LIN {X 0,Y 431.74,Z 953.951,A -85,B 0,C 180,E1 3788.335,E2 3788.335} C_VEL
LIN {X 0,Y 438.13,Z 926.777,A -85,B 0,C 180,E1 3787.877,E2 3787.877} C_VEL
LIN {X 0,Y 442.587,Z 899.79,A -85,B 0,C 180,E1 3787.482,E2 3787.482} C_VEL
LIN {X 0,Y 459.904,Z 746.935,A -85,B 0,C 180,E1 3785.438,E2 3785.438} C_VEL
LIN {X 0,Y 462.106,Z 727.315,A -85,B 0,C 180,E1 3785.152,E2 3785.152} C_VEL
LIN {X 0,Y 460.748,Z 722.782,A -85,B 0,C 180,E1 3780.497,E2 3780.497} C_VEL
LIN {X 0,Y 460.764,Z 722.91,A -85,B 0,C 180,E1 3779.005,E2 3779.005} C_VEL
LIN {X 0,Y 462.101,Z 727.286,A -85,B 0,C 180,E1 3774.661,E2 3774.661} C_VEL
LIN {X 0,Y 442.705,Z 898.388,A -85,B 0,C 180,E1 3772.376,E2 3772.376} C_VEL
LIN {X 0,Y 438.374,Z 924.66,A -85,B 0,C 180,E1 3771.993,E2 3771.993} C_VEL
LIN {X 0,Y 432.03,Z 951.964,A -85,B 0,C 180,E1 3771.518,E2 3771.518} C_VEL
LIN {X 0,Y 425.902,Z 973.345,A -85,B 0,C 180,E1 3771.046,E2 3771.046} C_VEL
LIN {X 0,Y 419.197,Z 993.326,A -85,B 0,C 180,E1 3770.513,E2 3770.513} C_VEL
LIN {X 0,Y 411.382,Z 1013.618,A -85,B 0,C 180,E1 3769.866,E2 3769.866} C_VEL
LIN {X 0,Y 401.355,Z 1036.487,A -85,B 0,C 180,E1 3768.989,E2 3768.989} C_VEL
LIN {X 0,Y 388.724,Z 1061.334,A -85,B 0,C 180,E1 3767.816,E2 3767.816} C_VEL
LIN {X 0,Y 378.046,Z 1080.059,A -85,B 0,C 180,E1 3766.742,E2 3766.742} C_VEL
LIN {X 0,Y 367.06,Z 1097.609,A -85,B 0,C 180,E1 3765.565,E2 3765.565} C_VEL
LIN {X 0,Y 355.375,Z 1114.731,A -85,B 0,C 180,E1 3764.215,E2 3764.215} C_VEL
LIN {X 0,Y 342.365,Z 1132.293,A -85,B 0,C 180,E1 3762.566,E2 3762.566} C_VEL
LIN {X 0,Y 325.314,Z 1153.259,A -85,B 0,C 180,E1 3760.147,E2 3760.147} C_VEL
LIN {X 0,Y 310.967,Z 1169.357,A -85,B 0,C 180,E1 3757.833,E2 3757.833} C_VEL
LIN {X 0,Y 297.909,Z 1183.077,A -85,B 0,C 180,E1 3755.454,E2 3755.454} C_VEL
LIN {X 0,Y 284.669,Z 1196.186,A -85,B 0,C 180,E1 3752.712,E2 3752.712} C_VEL
LIN {X 0,Y 270.089,Z 1209.874,A -85,B 0,C 180,E1 3749.198,E2 3749.198} C_VEL
LIN {X 0,Y 254.111,Z 1223.984,A -85,B 0,C 180,E1 3744.547,E2 3744.547} C_VEL
LIN {X 0,Y 242.024,Z 1234.259,A -85,B 0,C 180,E1 3740.221,E2 3740.221} C_VEL
LIN {X 0,Y 231.488,Z 1243.083,A -85,B 0,C 180,E1 3735.593,E2 3735.593} C_VEL
LIN {X 0,Y 221.707,Z 1251.328,A -85,B 0,C 180,E1 3730.167,E2 3730.167} C_VEL
LIN {X 0,Y 211.776,Z 1260.022,A -85,B 0,C 180,E1 3722.572,E2 3722.572} C_VEL
LIN {X 0,Y 206.37,Z 1265.193,A -85,B 0,C 180,E1 3716.479,E2 3716.479} C_VEL
LIN {X 0,Y 202.92,Z 1269.061,A -85,B 0,C 180,E1 3710.486,E2 3710.486} C_VEL
LIN {X 0,Y 200.916,Z 1271.91,A -85,B 0,C 180,E1 3704.416,E2 3704.416} C_VEL
LIN {X 0,Y 200.12,Z 1273.63,A -85,B 0,C 180,E1 3698.918,E2 3698.918} C_VEL
LIN {X 0,Y 199.932,Z 1274.524,A -85,B 0,C 180,E1 3693.736,E2 3693.736} C_VEL
LIN {X 0,Y 199.902,Z 1274.714,A -85,B 0,C 180,E1 3688.575,E2 3688.575} C_VEL
LIN {X 0,Y 200.031,Z 1274.064,A -85,B 0,C 180,E1 3682.83,E2 3682.83} C_VEL
LIN {X 0,Y 200.717,Z 1272.303,A -85,B 0,C 180,E1 3676.468,E2 3676.468} C_VEL
LIN {X 0,Y 202.505,Z 1269.613,A -85,B 0,C 180,E1 3670.391,E2 3670.391} C_VEL
LIN {X 0,Y 205.725,Z 1265.905,A -85,B 0,C 180,E1 3664.38,E2 3664.38} C_VEL
LIN {X 0,Y 210.576,Z 1261.15,A -85,B 0,C 180,E1 3658.523,E2 3658.523} C_VEL
LIN {X 0,Y 217.466,Z 1255.015,A -85,B 0,C 180,E1 3652.644,E2 3652.644} C_VEL
LIN {X 0,Y 227.949,Z 1246.234,A -85,B 0,C 180,E1 3646.14,E2 3646.14} C_VEL
LIN {X 0,Y 240.257,Z 1235.835,A -85,B 0,C 180,E1 3640.408,E2 3640.408} C_VEL
LIN {X 0,Y 251.535,Z 1226.259,A -85,B 0,C 180,E1 3636.215,E2 3636.215} C_VEL
LIN {X 0,Y 263.975,Z 1215.419,A -85,B 0,C 180,E1 3632.378,E2 3632.378} C_VEL
LIN {X 0,Y 279.527,Z 1201.327,A -85,B 0,C 180,E1 3628.38,E2 3628.38} C_VEL
LIN {X 0,Y 295.48,Z 1185.719,A -85,B 0,C 180,E1 3624.939,E2 3624.939} C_VEL
LIN {X 0,Y 309.223,Z 1171.411,A -85,B 0,C 180,E1 3622.383,E2 3622.383} C_VEL
LIN {X 0,Y 322.706,Z 1156.426,A -85,B 0,C 180,E1 3620.166,E2 3620.166} C_VEL
LIN {X 0,Y 337.881,Z 1138.297,A -85,B 0,C 180,E1 3617.958,E2 3617.958} C_VEL
LIN {X 0,Y 353.624,Z 1117.498,A -85,B 0,C 180,E1 3615.919,E2 3615.919} C_VEL
LIN {X 0,Y 366.029,Z 1099.508,A -85,B 0,C 180,E1 3614.472,E2 3614.472} C_VEL
LIN {X 0,Y 377.002,Z 1082.144,A -85,B 0,C 180,E1 3613.285,E2 3613.285} C_VEL
LIN {X 0,Y 387.675,Z 1063.625,A -85,B 0,C 180,E1 3612.206,E2 3612.206} C_VEL
LIN {X 0,Y 398.484,Z 1042.855,A -85,B 0,C 180,E1 3611.19,E2 3611.19} C_VEL
LIN {X 0,Y 410.324,Z 1016.781,A -85,B 0,C 180,E1 3610.147,E2 3610.147} C_VEL
LIN {X 0,Y 418.595,Z 995.638,A -85,B 0,C 180,E1 3609.458,E2 3609.458} C_VEL
LIN {X 0,Y 425.76,Z 974.544,A -85,B 0,C 180,E1 3608.889,E2 3608.889} C_VEL
LIN {X 0,Y 431.831,Z 953.572,A -85,B 0,C 180,E1 3608.419,E2 3608.419} C_VEL
LIN {X 0,Y 437.526,Z 929.769,A -85,B 0,C 180,E1 3607.991,E2 3607.991} C_VEL
LIN {X 0,Y 442.669,Z 900.46,A -85,B 0,C 180,E1 3607.558,E2 3607.558} C_VEL
LIN {X 0,Y 450.513,Z 832.504,A -85,B 0,C 180,E1 3606.642,E2 3606.642} C_VEL
LIN {X 0,Y 460.523,Z 743.446,A -85,B 0,C 180,E1 3605.461,E2 3605.461} C_VEL
LIN {X 0,Y 460.776,Z 740.62,A -85,B 0,C 180,E1 3605.335,E2 3605.335} C_VEL
LIN {X 0,Y 460.899,Z 737.599,A -85,B 0,C 180,E1 3604.988,E2 3604.988} C_VEL
LIN {X 0,Y 460.834,Z 734.987,A -85,B 0,C 180,E1 3604.394,E2 3604.394} C_VEL
LIN {X 0,Y 460.538,Z 733.277,A -85,B 0,C 180,E1 3603.464,E2 3603.464} C_VEL
LIN {X 0,Y 460.018,Z 731.722,A -85,B 0,C 180,E1 3601.278,E2 3601.278} C_VEL
LIN {X 0,Y 460.029,Z 730.802,A -85,B 0,C 180,E1 3600.249,E2 3600.249} C_VEL
LIN {X 0,Y 460.02,Z 731.113,A -85,B 0,C 180,E1 3599.377,E2 3599.377} C_VEL
LIN {X 0,Y 460.869,Z 734.659,A -85,B 0,C 180,E1 3595.723,E2 3595.723} C_VEL
LIN {X 0,Y 441.878,Z 899.528,A -85,B 0,C 180,E1 3593.558,E2 3593.558} C_VEL
LIN {X 0,Y 437.515,Z 925.726,A -85,B 0,C 180,E1 3593.185,E2 3593.185} C_VEL
LIN {X 0,Y 431.017,Z 953.376,A -85,B 0,C 180,E1 3592.738,E2 3592.738} C_VEL
LIN {X 0,Y 424.735,Z 974.983,A -85,B 0,C 180,E1 3592.299,E2 3592.299} C_VEL
LIN {X 0,Y 417.681,Z 995.66,A -85,B 0,C 180,E1 3591.784,E2 3591.784} C_VEL
LIN {X 0,Y 409.113,Z 1017.445,A -85,B 0,C 180,E1 3591.126,E2 3591.126} C_VEL
LIN {X 0,Y 396.795,Z 1044.344,A -85,B 0,C 180,E1 3590.119,E2 3590.119} C_VEL
LIN {X 0,Y 385.804,Z 1065.218,A -85,B 0,C 180,E1 3589.153,E2 3589.153} C_VEL
LIN {X 0,Y 375.409,Z 1083.081,A -85,B 0,C 180,E1 3588.165,E2 3588.165} C_VEL
LIN {X 0,Y 364.197,Z 1100.645,A -85,B 0,C 180,E1 3587.036,E2 3587.036} C_VEL
LIN {X 0,Y 351.419,Z 1118.995,A -85,B 0,C 180,E1 3585.625,E2 3585.625} C_VEL
LIN {X 0,Y 334.598,Z 1140.901,A -85,B 0,C 180,E1 3583.561,E2 3583.561} C_VEL
LIN {X 0,Y 319.494,Z 1158.677,A -85,B 0,C 180,E1 3581.466,E2 3581.466} C_VEL
LIN {X 0,Y 305.767,Z 1173.69,A -85,B 0,C 180,E1 3579.319,E2 3579.319} C_VEL
LIN {X 0,Y 292.283,Z 1187.492,A -85,B 0,C 180,E1 3576.94,E2 3576.94} C_VEL
LIN {X 0,Y 275.5,Z 1203.679,A -85,B 0,C 180,E1 3573.486,E2 3573.486} C_VEL
LIN {X 0,Y 258.969,Z 1218.346,A -85,B 0,C 180,E1 3569.413,E2 3569.413} C_VEL
LIN {X 0,Y 246.052,Z 1229.349,A -85,B 0,C 180,E1 3565.566,E2 3565.566} C_VEL
LIN {X 0,Y 233.713,Z 1239.549,A -85,B 0,C 180,E1 3561.122,E2 3561.122} C_VEL
LIN {X 0,Y 220.194,Z 1250.61,A -85,B 0,C 180,E1 3554.896,E2 3554.896} C_VEL
LIN {X 0,Y 209.957,Z 1258.964,A -85,B 0,C 180,E1 3548.587,E2 3548.587} C_VEL
LIN {X 0,Y 203.046,Z 1264.948,A -85,B 0,C 180,E1 3542.787,E2 3542.787} C_VEL
LIN {X 0,Y 198.108,Z 1269.63,A -85,B 0,C 180,E1 3537.006,E2 3537.006} C_VEL
LIN {X 0,Y 194.66,Z 1273.485,A -85,B 0,C 180,E1 3530.793,E2 3530.793} C_VEL
LIN {X 0,Y 192.709,Z 1276.35,A -85,B 0,C 180,E1 3524.412,E2 3524.412} C_VEL
LIN {X 0,Y 192.018,Z 1278.03,A -85,B 0,C 180,E1 3518.676,E2 3518.676} C_VEL
LIN {X 0,Y 191.915,Z 1278.81,A -85,B 0,C 180,E1 3513.875,E2 3513.875} C_VEL
LIN {X 0,Y 191.904,Z 1278.991,A -85,B 0,C 180,E1 3508.499,E2 3508.499} C_VEL
LIN {X 0,Y 191.976,Z 1278.363,A -85,B 0,C 180,E1 3502.811,E2 3502.811} C_VEL
LIN {X 0,Y 192.612,Z 1276.532,A -85,B 0,C 180,E1 3496.11,E2 3496.11} C_VEL
LIN {X 0,Y 194.525,Z 1273.637,A -85,B 0,C 180,E1 3489.533,E2 3489.533} C_VEL
LIN {X 0,Y 197.914,Z 1269.796,A -85,B 0,C 180,E1 3483.272,E2 3483.272} C_VEL
LIN {X 0,Y 202.778,Z 1265.151,A -85,B 0,C 180,E1 3477.479,E2 3477.479} C_VEL
LIN {X 0,Y 209.608,Z 1259.203,A -85,B 0,C 180,E1 3471.666,E2 3471.666} C_VEL
LIN {X 0,Y 219.533,Z 1251.054,A -85,B 0,C 180,E1 3465.452,E2 3465.452} C_VEL
LIN {X 0,Y 233.238,Z 1239.865,A -85,B 0,C 180,E1 3459.064,E2 3459.064} C_VEL
LIN {X 0,Y 245.459,Z 1229.753,A -85,B 0,C 180,E1 3454.62,E2 3454.62} C_VEL
LIN {X 0,Y 257.657,Z 1219.369,A -85,B 0,C 180,E1 3450.94,E2 3450.94} C_VEL
LIN {X 0,Y 271.539,Z 1207.058,A -85,B 0,C 180,E1 3447.406,E2 3447.406} C_VEL
LIN {X 0,Y 289.256,Z 1190.394,A -85,B 0,C 180,E1 3443.638,E2 3443.638} C_VEL
LIN {X 0,Y 304.892,Z 1174.436,A -85,B 0,C 180,E1 3440.82,E2 3440.82} C_VEL
LIN {X 0,Y 317.875,Z 1160.292,A -85,B 0,C 180,E1 3438.764,E2 3438.764} C_VEL
LIN {X 0,Y 331.232,Z 1144.698,A -85,B 0,C 180,E1 3436.87,E2 3436.87} C_VEL
LIN {X 0,Y 345.798,Z 1126.332,A -85,B 0,C 180,E1 3435.025,E2 3435.025} C_VEL
LIN {X 0,Y 361.963,Z 1103.695,A -85,B 0,C 180,E1 3433.193,E2 3433.193} C_VEL
LIN {X 0,Y 374.083,Z 1084.888,A -85,B 0,C 180,E1 3431.954,E2 3431.954} C_VEL
LIN {X 0,Y 384.933,Z 1066.371,A -85,B 0,C 180,E1 3430.916,E2 3430.916} C_VEL
LIN {X 0,Y 395.243,Z 1046.946,A -85,B 0,C 180,E1 3430.002,E2 3430.002} C_VEL
LIN {X 0,Y 406.787,Z 1022.539,A -85,B 0,C 180,E1 3429.051,E2 3429.051} C_VEL
LIN {X 0,Y 416.726,Z 997.638,A -85,B 0,C 180,E1 3428.277,E2 3428.277} C_VEL
LIN {X 0,Y 424.08,Z 976.293,A -85,B 0,C 180,E1 3427.737,E2 3427.737} C_VEL
LIN {X 0,Y 430.349,Z 954.947,A -85,B 0,C 180,E1 3427.296,E2 3427.296} C_VEL
LIN {X 0,Y 436.238,Z 930.604,A -85,B 0,C 180,E1 3426.893,E2 3426.893} C_VEL
LIN {X 0,Y 441.366,Z 901.504,A -85,B 0,C 180,E1 3426.473,E2 3426.473} C_VEL
LIN {X 0,Y 449.589,Z 831.186,A -85,B 0,C 180,E1 3425.54,E2 3425.54} C_VEL
LIN {X 0,Y 460.644,Z 734.296,A -85,B 0,C 180,E1 3424.264,E2 3424.264} C_VEL
LIN {X 0,Y 459.764,Z 730.724,A -85,B 0,C 180,E1 3420.374,E2 3420.374} C_VEL
LIN {X 0,Y 459.779,Z 730.934,A -85,B 0,C 180,E1 3419.003,E2 3419.003} C_VEL
LIN {X 0,Y 460.604,Z 734.521,A -85,B 0,C 180,E1 3415.558,E2 3415.558} C_VEL
LIN {X 0,Y 441.721,Z 898.431,A -85,B 0,C 180,E1 3413.408,E2 3413.408} C_VEL
LIN {X 0,Y 437.36,Z 924.593,A -85,B 0,C 180,E1 3413.037,E2 3413.037} C_VEL
LIN {X 0,Y 430.918,Z 952.063,A -85,B 0,C 180,E1 3412.575,E2 3412.575} C_VEL
LIN {X 0,Y 424.724,Z 973.443,A -85,B 0,C 180,E1 3412.118,E2 3412.118} C_VEL
LIN {X 0,Y 417.756,Z 993.938,A -85,B 0,C 180,E1 3411.589,E2 3411.589} C_VEL
LIN {X 0,Y 409.574,Z 1014.842,A -85,B 0,C 180,E1 3410.94,E2 3410.94} C_VEL
LIN {X 0,Y 398.51,Z 1039.526,A -85,B 0,C 180,E1 3410.009,E2 3410.009} C_VEL
LIN {X 0,Y 386.179,Z 1063.046,A -85,B 0,C 180,E1 3408.91,E2 3408.91} C_VEL
LIN {X 0,Y 375.176,Z 1081.917,A -85,B 0,C 180,E1 3407.846,E2 3407.846} C_VEL
LIN {X 0,Y 363.777,Z 1099.699,A -85,B 0,C 180,E1 3406.667,E2 3406.667} C_VEL
LIN {X 0,Y 349.753,Z 1119.674,A -85,B 0,C 180,E1 3405.088,E2 3405.088} C_VEL
LIN {X 0,Y 333.045,Z 1140.984,A -85,B 0,C 180,E1 3402.991,E2 3402.991} C_VEL
LIN {X 0,Y 319.288,Z 1157.039,A -85,B 0,C 180,E1 3401.049,E2 3401.049} C_VEL
LIN {X 0,Y 305.868,Z 1171.616,A -85,B 0,C 180,E1 3398.925,E2 3398.925} C_VEL
LIN {X 0,Y 291.356,Z 1186.35,A -85,B 0,C 180,E1 3396.326,E2 3396.326} C_VEL
LIN {X 0,Y 272.934,Z 1203.659,A -85,B 0,C 180,E1 3392.452,E2 3392.452} C_VEL
LIN {X 0,Y 259.083,Z 1215.825,A -85,B 0,C 180,E1 3388.964,E2 3388.964} C_VEL
LIN {X 0,Y 246.838,Z 1226.12,A -85,B 0,C 180,E1 3385.324,E2 3385.324} C_VEL
LIN {X 0,Y 235.057,Z 1235.716,A -85,B 0,C 180,E1 3381.126,E2 3381.126} C_VEL
LIN {X 0,Y 222.128,Z 1246.132,A -85,B 0,C 180,E1 3375.342,E2 3375.342} C_VEL
LIN {X 0,Y 211.001,Z 1254.958,A -85,B 0,C 180,E1 3368.728,E2 3368.728} C_VEL
LIN {X 0,Y 203.616,Z 1261.118,A -85,B 0,C 180,E1 3362.703,E2 3362.703} C_VEL
LIN {X 0,Y 198.359,Z 1265.894,A -85,B 0,C 180,E1 3356.664,E2 3356.664} C_VEL
LIN {X 0,Y 194.841,Z 1269.623,A -85,B 0,C 180,E1 3350.432,E2 3350.432} C_VEL
LIN {X 0,Y 192.781,Z 1272.446,A -85,B 0,C 180,E1 3343.811,E2 3343.811} C_VEL
LIN {X 0,Y 192.022,Z 1274.252,A -85,B 0,C 180,E1 3336.887,E2 3336.887} C_VEL
LIN {X 0,Y 191.895,Z 1274.835,A -85,B 0,C 180,E1 3330.904,E2 3330.904} C_VEL
LIN {X 0,Y 191.948,Z 1274.558,A -85,B 0,C 180,E1 3325.228,E2 3325.228} C_VEL
LIN {X 0,Y 192.272,Z 1273.421,A -85,B 0,C 180,E1 3319.219,E2 3319.219} C_VEL
LIN {X 0,Y 193.959,Z 1270.803,A -85,B 0,C 180,E1 3311.681,E2 3311.681} C_VEL
LIN {X 0,Y 197.747,Z 1266.561,A -85,B 0,C 180,E1 3304.164,E2 3304.164} C_VEL
LIN {X 0,Y 202.958,Z 1261.742,A -85,B 0,C 180,E1 3297.866,E2 3297.866} C_VEL
LIN {X 0,Y 209.774,Z 1256.004,A -85,B 0,C 180,E1 3292.069,E2 3292.069} C_VEL
LIN {X 0,Y 218.741,Z 1248.794,A -85,B 0,C 180,E1 3286.364,E2 3286.364} C_VEL
LIN {X 0,Y 231.631,Z 1238.655,A -85,B 0,C 180,E1 3280.191,E2 3280.191} C_VEL
LIN {X 0,Y 245.442,Z 1227.37,A -85,B 0,C 180,E1 3275.047,E2 3275.047} C_VEL
LIN {X 0,Y 258.246,Z 1216.647,A -85,B 0,C 180,E1 3271.182,E2 3271.182} C_VEL
LIN {X 0,Y 271.332,Z 1205.201,A -85,B 0,C 180,E1 3267.837,E2 3267.837} C_VEL
LIN {X 0,Y 287.49,Z 1190.322,A -85,B 0,C 180,E1 3264.343,E2 3264.343} C_VEL
LIN {X 0,Y 304.56,Z 1173.182,A -85,B 0,C 180,E1 3261.212,E2 3261.212} C_VEL
LIN {X 0,Y 318.298,Z 1158.357,A -85,B 0,C 180,E1 3259.018,E2 3259.018} C_VEL
LIN {X 0,Y 331.617,Z 1142.926,A -85,B 0,C 180,E1 3257.121,E2 3257.121} C_VEL
LIN {X 0,Y 344.841,Z 1126.397,A -85,B 0,C 180,E1 3255.426,E2 3255.426} C_VEL
LIN {X 0,Y 360.541,Z 1104.918,A -85,B 0,C 180,E1 3253.612,E2 3253.612} C_VEL
LIN {X 0,Y 373.975,Z 1084.245,A -85,B 0,C 180,E1 3252.194,E2 3252.194} C_VEL
LIN {X 0,Y 385.128,Z 1065.328,A -85,B 0,C 180,E1 3251.109,E2 3251.109} C_VEL
LIN {X 0,Y 395.152,Z 1046.532,A -85,B 0,C 180,E1 3250.198,E2 3250.198} C_VEL
LIN {X 0,Y 405.276,Z 1025.348,A -85,B 0,C 180,E1 3249.336,E2 3249.336} C_VEL
LIN {X 0,Y 416.413,Z 998.283,A -85,B 0,C 180,E1 3248.438,E2 3248.438} C_VEL
LIN {X 0,Y 423.965,Z 976.595,A -85,B 0,C 180,E1 3247.862,E2 3247.862} C_VEL
LIN {X 0,Y 430.234,Z 955.468,A -85,B 0,C 180,E1 3247.397,E2 3247.397} C_VEL
LIN {X 0,Y 435.566,Z 933.878,A -85,B 0,C 180,E1 3247.012,E2 3247.012} C_VEL
LIN {X 0,Y 440.772,Z 907.08,A -85,B 0,C 180,E1 3246.616,E2 3246.616} C_VEL
LIN {X 0,Y 445.894,Z 865.845,A -85,B 0,C 180,E1 3246.062,E2 3246.062} C_VEL
LIN {X 0,Y 460.856,Z 734.46,A -85,B 0,C 180,E1 3244.324,E2 3244.324} C_VEL
LIN {X 0,Y 460.018,Z 731.722,A -85,B 0,C 180,E1 3241.278,E2 3241.278} C_VEL
LIN {X 0,Y 459.91,Z 731.875,A -85,B 0,C 180,E1 3240.524,E2 3240.524} C_VEL
LIN {X 0,Y 459.624,Z 734.239,A -85,B 0,C 180,E1 3239.525,E2 3239.525} C_VEL
LIN {X 0,Y 459.25,Z 740.324,A -85,B 0,C 180,E1 3237.684,E2 3237.684} C_VEL
LIN {X 0,Y 459.371,Z 741.488,A -85,B 0,C 180,E1 3236.99,E2 3236.99} C_VEL
LIN {X 0,Y 459.483,Z 741.921,A -85,B 0,C 180,E1 3236.627,E2 3236.627} C_VEL
LIN {X 0,Y 441.049,Z 899.462,A -85,B 0,C 180,E1 3234.596,E2 3234.596} C_VEL
LIN {X 0,Y 436.611,Z 925.784,A -85,B 0,C 180,E1 3234.23,E2 3234.23} C_VEL
LIN {X 0,Y 430.074,Z 953.299,A -85,B 0,C 180,E1 3233.801,E2 3233.801} C_VEL
LIN {X 0,Y 423.73,Z 974.904,A -85,B 0,C 180,E1 3233.379,E2 3233.379} C_VEL
LIN {X 0,Y 416.744,Z 995.196,A -85,B 0,C 180,E1 3232.894,E2 3232.894} C_VEL
LIN {X 0,Y 408.278,Z 1016.55,A -85,B 0,C 180,E1 3232.277,E2 3232.277} C_VEL
LIN {X 0,Y 396.414,Z 1042.456,A -85,B 0,C 180,E1 3231.354,E2 3231.354} C_VEL
LIN {X 0,Y 384.812,Z 1064.32,A -85,B 0,C 180,E1 3230.389,E2 3230.389} C_VEL
LIN {X 0,Y 373.799,Z 1083.021,A -85,B 0,C 180,E1 3229.394,E2 3229.394} C_VEL
LIN {X 0,Y 362.18,Z 1100.947,A -85,B 0,C 180,E1 3228.277,E2 3228.277} C_VEL
LIN {X 0,Y 348.576,Z 1120.129,A -85,B 0,C 180,E1 3226.837,E2 3226.837} C_VEL
LIN {X 0,Y 330.991,Z 1142.406,A -85,B 0,C 180,E1 3224.763,E2 3224.763} C_VEL
LIN {X 0,Y 316.949,Z 1158.589,A -85,B 0,C 180,E1 3222.891,E2 3222.891} C_VEL
LIN {X 0,Y 303.625,Z 1172.869,A -85,B 0,C 180,E1 3220.909,E2 3220.909} C_VEL
LIN {X 0,Y 289.345,Z 1187.167,A -85,B 0,C 180,E1 3218.512,E2 3218.512} C_VEL
LIN {X 0,Y 272.156,Z 1203.312,A -85,B 0,C 180,E1 3215.137,E2 3215.137} C_VEL
LIN {X 0,Y 255.487,Z 1217.679,A -85,B 0,C 180,E1 3211.224,E2 3211.224} C_VEL
LIN {X 0,Y 242.043,Z 1228.74,A -85,B 0,C 180,E1 3207.413,E2 3207.413} C_VEL
LIN {X 0,Y 229.696,Z 1238.533,A -85,B 0,C 180,E1 3203.207,E2 3203.207} C_VEL
LIN {X 0,Y 217.568,Z 1247.953,A -85,B 0,C 180,E1 3198.103,E2 3198.103} C_VEL
LIN {X 0,Y 204.373,Z 1258.177,A -85,B 0,C 180,E1 3190.682,E2 3190.682} C_VEL
LIN {X 0,Y 196.392,Z 1264.599,A -85,B 0,C 180,E1 3184.399,E2 3184.399} C_VEL
LIN {X 0,Y 190.756,Z 1269.54,A -85,B 0,C 180,E1 3178.137,E2 3178.137} C_VEL
LIN {X 0,Y 187.108,Z 1273.257,A -85,B 0,C 180,E1 3171.956,E2 3171.956} C_VEL
LIN {X 0,Y 184.964,Z 1276.029,A -85,B 0,C 180,E1 3165.672,E2 3165.672} C_VEL
LIN {X 0,Y 184.096,Z 1277.733,A -85,B 0,C 180,E1 3159.999,E2 3159.999} C_VEL
LIN {X 0,Y 183.918,Z 1278.699,A -85,B 0,C 180,E1 3154.356,E2 3154.356} C_VEL
LIN {X 0,Y 183.896,Z 1278.926,A -85,B 0,C 180,E1 3148.745,E2 3148.745} C_VEL
LIN {X 0,Y 183.975,Z 1278.344,A -85,B 0,C 180,E1 3142.81,E2 3142.81} C_VEL
LIN {X 0,Y 184.667,Z 1276.531,A -85,B 0,C 180,E1 3135.745,E2 3135.745} C_VEL
LIN {X 0,Y 186.7,Z 1273.709,A -85,B 0,C 180,E1 3128.964,E2 3128.964} C_VEL
LIN {X 0,Y 190.323,Z 1269.914,A -85,B 0,C 180,E1 3122.455,E2 3122.455} C_VEL
LIN {X 0,Y 195.791,Z 1265.059,A -85,B 0,C 180,E1 3116.167,E2 3116.167} C_VEL
LIN {X 0,Y 203.144,Z 1259.07,A -85,B 0,C 180,E1 3110.161,E2 3110.161} C_VEL
LIN {X 0,Y 213.708,Z 1250.898,A -85,B 0,C 180,E1 3103.825,E2 3103.825} C_VEL
LIN {X 0,Y 227.972,Z 1239.815,A -85,B 0,C 180,E1 3097.443,E2 3097.443} C_VEL
LIN {X 0,Y 240.89,Z 1229.572,A -85,B 0,C 180,E1 3092.94,E2 3092.94} C_VEL
LIN {X 0,Y 253.57,Z 1219.161,A -85,B 0,C 180,E1 3089.273,E2 3089.273} C_VEL
LIN {X 0,Y 267.725,Z 1207.011,A -85,B 0,C 180,E1 3085.823,E2 3085.823} C_VEL
LIN {X 0,Y 285.218,Z 1191.075,A -85,B 0,C 180,E1 3082.247,E2 3082.247} C_VEL
LIN {X 0,Y 302.024,Z 1174.342,A -85,B 0,C 180,E1 3079.339,E2 3079.339} C_VEL
LIN {X 0,Y 315.72,Z 1159.733,A -85,B 0,C 180,E1 3077.274,E2 3077.274} C_VEL
LIN {X 0,Y 329.354,Z 1144.095,A -85,B 0,C 180,E1 3075.433,E2 3075.433} C_VEL
LIN {X 0,Y 345.517,Z 1124.009,A -85,B 0,C 180,E1 3073.496,E2 3073.496} C_VEL
LIN {X 0,Y 361.079,Z 1102.252,A -85,B 0,C 180,E1 3071.825,E2 3071.825} C_VEL
LIN {X 0,Y 373.17,Z 1083.664,A -85,B 0,C 180,E1 3070.654,E2 3070.654} C_VEL
LIN {X 0,Y 383.931,Z 1065.464,A -85,B 0,C 180,E1 3069.677,E2 3069.677} C_VEL
LIN {X 0,Y 394.591,Z 1045.533,A -85,B 0,C 180,E1 3068.78,E2 3068.78} C_VEL
LIN {X 0,Y 406.756,Z 1019.651,A -85,B 0,C 180,E1 3067.829,E2 3067.829} C_VEL
LIN {X 0,Y 415.925,Z 996.763,A -85,B 0,C 180,E1 3067.153,E2 3067.153} C_VEL
LIN {X 0,Y 423.147,Z 975.956,A -85,B 0,C 180,E1 3066.649,E2 3066.649} C_VEL
LIN {X 0,Y 429.583,Z 954.188,A -85,B 0,C 180,E1 3066.219,E2 3066.219} C_VEL
LIN {X 0,Y 436.049,Z 927.425,A -85,B 0,C 180,E1 3065.797,E2 3065.797} C_VEL
LIN {X 0,Y 440.737,Z 899.893,A -85,B 0,C 180,E1 3065.413,E2 3065.413} C_VEL
LIN {X 0,Y 455.47,Z 774.09,A -85,B 0,C 180,E1 3063.787,E2 3063.787} C_VEL
LIN {X 0,Y 459.263,Z 741.532,A -85,B 0,C 180,E1 3063.37,E2 3063.37} C_VEL
LIN {X 0,Y 458.789,Z 738.665,A -85,B 0,C 180,E1 3060.375,E2 3060.375} C_VEL
LIN {X 0,Y 458.794,Z 738.956,A -85,B 0,C 180,E1 3059.001,E2 3059.001} C_VEL
LIN {X 0,Y 459.236,Z 741.61,A -85,B 0,C 180,E1 3056.466,E2 3056.466} C_VEL
LIN {X 0,Y 440.864,Z 898.602,A -85,B 0,C 180,E1 3054.443,E2 3054.443} C_VEL
LIN {X 0,Y 436.375,Z 925.165,A -85,B 0,C 180,E1 3054.075,E2 3054.075} C_VEL
LIN {X 0,Y 429.894,Z 952.378,A -85,B 0,C 180,E1 3053.633,E2 3053.633} C_VEL
LIN {X 0,Y 423.695,Z 973.54,A -85,B 0,C 180,E1 3053.197,E2 3053.197} C_VEL
LIN {X 0,Y 416.775,Z 993.702,A -85,B 0,C 180,E1 3052.695,E2 3052.695} C_VEL
LIN {X 0,Y 408.847,Z 1013.809,A -85,B 0,C 180,E1 3052.097,E2 3052.097} C_VEL
LIN {X 0,Y 398.575,Z 1036.678,A -85,B 0,C 180,E1 3051.278,E2 3051.278} C_VEL
LIN {X 0,Y 385.617,Z 1061.522,A -85,B 0,C 180,E1 3050.181,E2 3050.181} C_VEL
LIN {X 0,Y 373.985,Z 1081.3,A -85,B 0,C 180,E1 3049.111,E2 3049.111} C_VEL
LIN {X 0,Y 362.871,Z 1098.462,A -85,B 0,C 180,E1 3048.023,E2 3048.023} C_VEL
LIN {X 0,Y 350.376,Z 1116.131,A -85,B 0,C 180,E1 3046.697,E2 3046.697} C_VEL
LIN {X 0,Y 334.184,Z 1137.041,A -85,B 0,C 180,E1 3044.79,E2 3044.79} C_VEL
LIN {X 0,Y 317.656,Z 1156.082,A -85,B 0,C 180,E1 3042.6,E2 3042.6} C_VEL
LIN {X 0,Y 304.269,Z 1170.385,A -85,B 0,C 180,E1 3040.594,E2 3040.594} C_VEL
LIN {X 0,Y 290.589,Z 1184.031,A -85,B 0,C 180,E1 3038.295,E2 3038.295} C_VEL
LIN {X 0,Y 275.893,Z 1197.766,A -85,B 0,C 180,E1 3035.468,E2 3035.468} C_VEL
LIN {X 0,Y 257.22,Z 1213.999,A -85,B 0,C 180,E1 3031.182,E2 3031.182} C_VEL
LIN {X 0,Y 242.821,Z 1225.703,A -85,B 0,C 180,E1 3027.152,E2 3027.152} C_VEL
LIN {X 0,Y 230.475,Z 1235.355,A -85,B 0,C 180,E1 3022.973,E2 3022.973} C_VEL
LIN {X 0,Y 218.331,Z 1244.621,A -85,B 0,C 180,E1 3017.903,E2 3017.903} C_VEL
LIN {X 0,Y 204.947,Z 1254.752,A -85,B 0,C 180,E1 3010.465,E2 3010.465} C_VEL
LIN {X 0,Y 196.979,Z 1260.958,A -85,B 0,C 180,E1 3004.303,E2 3004.303} C_VEL
LIN {X 0,Y 191.229,Z 1265.782,A -85,B 0,C 180,E1 2998.081,E2 2998.081} C_VEL
LIN {X 0,Y 187.311,Z 1269.556,A -85,B 0,C 180,E1 2991.621,E2 2991.621} C_VEL
LIN {X 0,Y 185.029,Z 1272.312,A -85,B 0,C 180,E1 2985.042,E2 2985.042} C_VEL
LIN {X 0,Y 184.131,Z 1273.94,A -85,B 0,C 180,E1 2979.069,E2 2979.069} C_VEL
LIN {X 0,Y 183.933,Z 1274.722,A -85,B 0,C 180,E1 2973.749,E2 2973.749} C_VEL
LIN {X 0,Y 183.905,Z 1274.889,A -85,B 0,C 180,E1 2968.451,E2 2968.451} C_VEL
LIN {X 0,Y 184.046,Z 1274.307,A -85,B 0,C 180,E1 2962.517,E2 2962.517} C_VEL
LIN {X 0,Y 184.898,Z 1272.543,A -85,B 0,C 180,E1 2955.466,E2 2955.466} C_VEL
LIN {X 0,Y 187.12,Z 1269.792,A -85,B 0,C 180,E1 2948.704,E2 2948.704} C_VEL
LIN {X 0,Y 190.93,Z 1266.085,A -85,B 0,C 180,E1 2942.231,E2 2942.231} C_VEL
LIN {X 0,Y 196.263,Z 1261.581,A -85,B 0,C 180,E1 2936.28,E2 2936.28} C_VEL
LIN {X 0,Y 203.64,Z 1255.794,A -85,B 0,C 180,E1 2930.347,E2 2930.347} C_VEL
LIN {X 0,Y 213.235,Z 1248.535,A -85,B 0,C 180,E1 2924.555,E2 2924.555} C_VEL
LIN {X 0,Y 227.432,Z 1237.836,A -85,B 0,C 180,E1 2918.113,E2 2918.113} C_VEL
LIN {X 0,Y 241.366,Z 1226.949,A -85,B 0,C 180,E1 2913.212,E2 2913.212} C_VEL
LIN {X 0,Y 254.702,Z 1216.168,A -85,B 0,C 180,E1 2909.384,E2 2909.384} C_VEL
LIN {X 0,Y 269.004,Z 1204.029,A -85,B 0,C 180,E1 2905.925,E2 2905.925} C_VEL
LIN {X 0,Y 288.063,Z 1186.663,A -85,B 0,C 180,E1 2902.084,E2 2902.084} C_VEL
LIN {X 0,Y 302.47,Z 1172.429,A -85,B 0,C 180,E1 2899.61,E2 2899.61} C_VEL
LIN {X 0,Y 316.535,Z 1157.522,A -85,B 0,C 180,E1 2897.477,E2 2897.477} C_VEL
LIN {X 0,Y 330.567,Z 1141.499,A -85,B 0,C 180,E1 2895.58,E2 2895.58} C_VEL
LIN {X 0,Y 347.024,Z 1121.034,A -85,B 0,C 180,E1 2893.604,E2 2893.604} C_VEL
LIN {X 0,Y 361.829,Z 1100.344,A -85,B 0,C 180,E1 2892.005,E2 2892.005} C_VEL
LIN {X 0,Y 373.587,Z 1082.313,A -85,B 0,C 180,E1 2890.847,E2 2890.847} C_VEL
LIN {X 0,Y 384.56,Z 1063.793,A -85,B 0,C 180,E1 2889.833,E2 2889.833} C_VEL
LIN {X 0,Y 395.654,Z 1043.021,A -85,B 0,C 180,E1 2888.883,E2 2888.883} C_VEL
LIN {X 0,Y 408.053,Z 1016.298,A -85,B 0,C 180,E1 2887.887,E2 2887.887} C_VEL
LIN {X 0,Y 416.72,Z 994.516,A -85,B 0,C 180,E1 2887.232,E2 2887.232} C_VEL
LIN {X 0,Y 423.814,Z 973.941,A -85,B 0,C 180,E1 2886.718,E2 2886.718} C_VEL
LIN {X 0,Y 430.142,Z 952.377,A -85,B 0,C 180,E1 2886.272,E2 2886.272} C_VEL
LIN {X 0,Y 436.629,Z 925.144,A -85,B 0,C 180,E1 2885.83,E2 2885.83} C_VEL
LIN {X 0,Y 441.116,Z 898.612,A -85,B 0,C 180,E1 2885.463,E2 2885.463} C_VEL
LIN {X 0,Y 459.485,Z 741.738,A -85,B 0,C 180,E1 2883.44,E2 2883.44} C_VEL
LIN {X 0,Y 459.051,Z 738.747,A -85,B 0,C 180,E1 2880.125,E2 2880.125} C_VEL
LIN {X 0,Y 459.031,Z 739.278,A -85,B 0,C 180,E1 2879.251,E2 2879.251} C_VEL
LIN {X 0,Y 459.371,Z 741.488,A -85,B 0,C 180,E1 2876.99,E2 2876.99} C_VEL
LIN {X 0,Y 459.317,Z 742.586,A -85,B 0,C 180,E1 2876.806,E2 2876.806} C_VEL
LIN {X 0,Y 458.963,Z 745.814,A -85,B 0,C 180,E1 2876.713,E2 2876.713} C_VEL
LIN {X 0,Y 458.316,Z 750.653,A -85,B 0,C 180,E1 2876.827,E2 2876.827} C_VEL
LIN {X 0,Y 456.914,Z 760.483,A -85,B 0,C 180,E1 2877.289,E2 2877.289} C_VEL
LIN {X 0,Y 456.324,Z 765.132,A -85,B 0,C 180,E1 2877.338,E2 2877.338} C_VEL
LIN {X 0,Y 440.335,Z 899.61,A -85,B 0,C 180,E1 2875.634,E2 2875.634} C_VEL
LIN {X 0,Y 435.66,Z 926.874,A -85,B 0,C 180,E1 2875.265,E2 2875.265} C_VEL
LIN {X 0,Y 429.099,Z 953.873,A -85,B 0,C 180,E1 2874.857,E2 2874.857} C_VEL
LIN {X 0,Y 422.877,Z 974.825,A -85,B 0,C 180,E1 2874.464,E2 2874.464} C_VEL
LIN {X 0,Y 415.69,Z 995.469,A -85,B 0,C 180,E1 2873.99,E2 2873.99} C_VEL
LIN {X 0,Y 407.061,Z 1016.962,A -85,B 0,C 180,E1 2873.392,E2 2873.392} C_VEL
LIN {X 0,Y 394.758,Z 1043.357,A -85,B 0,C 180,E1 2872.481,E2 2872.481} C_VEL
LIN {X 0,Y 383.534,Z 1064.235,A -85,B 0,C 180,E1 2871.591,E2 2871.591} C_VEL
LIN {X 0,Y 372.328,Z 1083.014,A -85,B 0,C 180,E1 2870.629,E2 2870.629} C_VEL
LIN {X 0,Y 359.951,Z 1101.812,A -85,B 0,C 180,E1 2869.493,E2 2869.493} C_VEL
LIN {X 0,Y 344.093,Z 1123.679,A -85,B 0,C 180,E1 2867.875,E2 2867.875} C_VEL
LIN {X 0,Y 327.647,Z 1143.778,A -85,B 0,C 180,E1 2866.004,E2 2866.004} C_VEL
LIN {X 0,Y 313.743,Z 1159.431,A -85,B 0,C 180,E1 2864.223,E2 2864.223} C_VEL
LIN {X 0,Y 300.16,Z 1173.63,A -85,B 0,C 180,E1 2862.284,E2 2862.284} C_VEL
LIN {X 0,Y 285.328,Z 1188.089,A -85,B 0,C 180,E1 2859.887,E2 2859.887} C_VEL
LIN {X 0,Y 266.429,Z 1205.162,A -85,B 0,C 180,E1 2856.286,E2 2856.286} C_VEL
LIN {X 0,Y 250.74,Z 1218.233,A -85,B 0,C 180,E1 2852.704,E2 2852.704} C_VEL
LIN {X 0,Y 236.943,Z 1229.168,A -85,B 0,C 180,E1 2848.925,E2 2848.925} C_VEL
LIN {X 0,Y 224.143,Z 1238.905,A -85,B 0,C 180,E1 2844.705,E2 2844.705} C_VEL
LIN {X 0,Y 209.917,Z 1249.497,A -85,B 0,C 180,E1 2838.801,E2 2838.801} C_VEL
LIN {X 0,Y 197.544,Z 1258.476,A -85,B 0,C 180,E1 2831.909,E2 2831.909} C_VEL
LIN {X 0,Y 189.252,Z 1264.749,A -85,B 0,C 180,E1 2825.546,E2 2825.546} C_VEL
LIN {X 0,Y 183.241,Z 1269.659,A -85,B 0,C 180,E1 2819.043,E2 2819.043} C_VEL
LIN {X 0,Y 179.182,Z 1273.492,A -85,B 0,C 180,E1 2812.289,E2 2812.289} C_VEL
LIN {X 0,Y 176.881,Z 1276.288,A -85,B 0,C 180,E1 2805.397,E2 2805.397} C_VEL
LIN {X 0,Y 176.018,Z 1278.012,A -85,B 0,C 180,E1 2798.724,E2 2798.724} C_VEL
LIN {X 0,Y 175.913,Z 1278.705,A -85,B 0,C 180,E1 2793.249,E2 2793.249} C_VEL
LIN {X 0,Y 175.912,Z 1278.793,A -85,B 0,C 180,E1 2788.036,E2 2788.036} C_VEL
LIN {X 0,Y 175.986,Z 1278.187,A -85,B 0,C 180,E1 2782.154,E2 2782.154} C_VEL
LIN {X 0,Y 176.749,Z 1276.494,A -85,B 0,C 180,E1 2775.243,E2 2775.243} C_VEL
LIN {X 0,Y 179.067,Z 1273.59,A -85,B 0,C 180,E1 2767.961,E2 2767.961} C_VEL
LIN {X 0,Y 183.01,Z 1269.823,A -85,B 0,C 180,E1 2761.254,E2 2761.254} C_VEL
LIN {X 0,Y 188.913,Z 1264.967,A -85,B 0,C 180,E1 2754.757,E2 2754.757} C_VEL
LIN {X 0,Y 196.72,Z 1259.018,A -85,B 0,C 180,E1 2748.633,E2 2748.633} C_VEL
LIN {X 0,Y 207.37,Z 1251.225,A -85,B 0,C 180,E1 2742.453,E2 2742.453} C_VEL
LIN {X 0,Y 222.956,Z 1239.722,A -85,B 0,C 180,E1 2735.726,E2 2735.726} C_VEL
LIN {X 0,Y 236.306,Z 1229.566,A -85,B 0,C 180,E1 2731.261,E2 2731.261} C_VEL
LIN {X 0,Y 249.423,Z 1219.181,A -85,B 0,C 180,E1 2727.623,E2 2727.623} C_VEL
LIN {X 0,Y 264.177,Z 1206.917,A -85,B 0,C 180,E1 2724.185,E2 2724.185} C_VEL
LIN {X 0,Y 282.151,Z 1190.98,A -85,B 0,C 180,E1 2720.671,E2 2720.671} C_VEL
LIN {X 0,Y 299.362,Z 1174.248,A -85,B 0,C 180,E1 2717.83,E2 2717.83} C_VEL
LIN {X 0,Y 313.215,Z 1159.787,A -85,B 0,C 180,E1 2715.84,E2 2715.84} C_VEL
LIN {X 0,Y 326.807,Z 1144.51,A -85,B 0,C 180,E1 2714.087,E2 2714.087} C_VEL
LIN {X 0,Y 341.887,Z 1126.144,A -85,B 0,C 180,E1 2712.35,E2 2712.35} C_VEL
LIN {X 0,Y 358.623,Z 1103.421,A -85,B 0,C 180,E1 2710.626,E2 2710.626} C_VEL
LIN {X 0,Y 371.259,Z 1084.339,A -85,B 0,C 180,E1 2709.456,E2 2709.456} C_VEL
LIN {X 0,Y 382.176,Z 1066.182,A -85,B 0,C 180,E1 2708.51,E2 2708.51} C_VEL
LIN {X 0,Y 392.489,Z 1047.242,A -85,B 0,C 180,E1 2707.681,E2 2707.681} C_VEL
LIN {X 0,Y 403.357,Z 1024.89,A -85,B 0,C 180,E1 2706.865,E2 2706.865} C_VEL
LIN {X 0,Y 414.304,Z 998.532,A -85,B 0,C 180,E1 2706.093,E2 2706.093} C_VEL
LIN {X 0,Y 422.117,Z 976.39,A -85,B 0,C 180,E1 2705.573,E2 2705.573} C_VEL
LIN {X 0,Y 428.492,Z 955.147,A -85,B 0,C 180,E1 2705.168,E2 2705.168} C_VEL
LIN {X 0,Y 434.27,Z 931.837,A -85,B 0,C 180,E1 2704.809,E2 2704.809} C_VEL
LIN {X 0,Y 439.769,Z 901.821,A -85,B 0,C 180,E1 2704.398,E2 2704.398} C_VEL
LIN {X 0,Y 447.506,Z 837.949,A -85,B 0,C 180,E1 2703.582,E2 2703.582} C_VEL
LIN {X 0,Y 457.992,Z 748.685,A -85,B 0,C 180,E1 2702.44,E2 2702.44} C_VEL
LIN {X 0,Y 457.806,Z 746.607,A -85,B 0,C 180,E1 2700.25,E2 2700.25} C_VEL
LIN {X 0,Y 457.812,Z 746.835,A -85,B 0,C 180,E1 2699.124,E2 2699.124} C_VEL
LIN {X 0,Y 457.97,Z 748.818,A -85,B 0,C 180,E1 2697.378,E2 2697.378} C_VEL
LIN {X 0,Y 440.155,Z 898.747,A -85,B 0,C 180,E1 2695.482,E2 2695.482} C_VEL
LIN {X 0,Y 435.572,Z 925.529,A -85,B 0,C 180,E1 2695.121,E2 2695.121} C_VEL
LIN {X 0,Y 429.047,Z 952.586,A -85,B 0,C 180,E1 2694.697,E2 2694.697} C_VEL
LIN {X 0,Y 422.817,Z 973.638,A -85,B 0,C 180,E1 2694.28,E2 2694.28} C_VEL
LIN {X 0,Y 415.665,Z 994.234,A -85,B 0,C 180,E1 2693.786,E2 2693.786} C_VEL
LIN {X 0,Y 407.341,Z 1015.033,A -85,B 0,C 180,E1 2693.187,E2 2693.187} C_VEL
LIN {X 0,Y 395.81,Z 1040.11,A -85,B 0,C 180,E1 2692.306,E2 2692.306} C_VEL
LIN {X 0,Y 383.381,Z 1063.234,A -85,B 0,C 180,E1 2691.299,E2 2691.299} C_VEL
LIN {X 0,Y 372.27,Z 1081.806,A -85,B 0,C 180,E1 2690.32,E2 2690.32} C_VEL
LIN {X 0,Y 360.804,Z 1099.222,A -85,B 0,C 180,E1 2689.25,E2 2689.25} C_VEL
LIN {X 0,Y 347.202,Z 1118.082,A -85,B 0,C 180,E1 2687.864,E2 2687.864} C_VEL
LIN {X 0,Y 329.033,Z 1140.667,A -85,B 0,C 180,E1 2685.799,E2 2685.799} C_VEL
LIN {X 0,Y 314.301,Z 1157.226,A -85,B 0,C 180,E1 2683.904,E2 2683.904} C_VEL
LIN {X 0,Y 300.776,Z 1171.32,A -85,B 0,C 180,E1 2681.956,E2 2681.956} C_VEL
LIN {X 0,Y 286.802,Z 1184.89,A -85,B 0,C 180,E1 2679.698,E2 2679.698} C_VEL
LIN {X 0,Y 269.45,Z 1200.645,A -85,B 0,C 180,E1 2676.44,E2 2676.44} C_VEL
LIN {X 0,Y 251.579,Z 1215.443,A -85,B 0,C 180,E1 2672.421,E2 2672.421} C_VEL
LIN {X 0,Y 237.713,Z 1226.306,A -85,B 0,C 180,E1 2668.645,E2 2668.645} C_VEL
LIN {X 0,Y 224.916,Z 1235.903,A -85,B 0,C 180,E1 2664.453,E2 2664.453} C_VEL
LIN {X 0,Y 210.682,Z 1246.318,A -85,B 0,C 180,E1 2658.587,E2 2658.587} C_VEL
LIN {X 0,Y 198.101,Z 1255.236,A -85,B 0,C 180,E1 2651.668,E2 2651.668} C_VEL
LIN {X 0,Y 189.824,Z 1261.301,A -85,B 0,C 180,E1 2645.418,E2 2645.418} C_VEL
LIN {X 0,Y 183.721,Z 1266.077,A -85,B 0,C 180,E1 2638.98,E2 2638.98} C_VEL
LIN {X 0,Y 179.536,Z 1269.804,A -85,B 0,C 180,E1 2632.263,E2 2632.263} C_VEL
LIN {X 0,Y 177.018,Z 1272.625,A -85,B 0,C 180,E1 2625.069,E2 2625.069} C_VEL
LIN {X 0,Y 176.071,Z 1274.295,A -85,B 0,C 180,E1 2618.171,E2 2618.171} C_VEL
LIN {X 0,Y 175.918,Z 1274.92,A -85,B 0,C 180,E1 2612.289,E2 2612.289} C_VEL
LIN {X 0,Y 175.922,Z 1274.887,A -85,B 0,C 180,E1 2607.077,E2 2607.077} C_VEL
LIN {X 0,Y 176.085,Z 1274.262,A -85,B 0,C 180,E1 2601.52,E2 2601.52} C_VEL
LIN {X 0,Y 177.071,Z 1272.569,A -85,B 0,C 180,E1 2594.62,E2 2594.62} C_VEL
LIN {X 0,Y 179.575,Z 1269.791,A -85,B 0,C 180,E1 2587.564,E2 2587.564} C_VEL
LIN {X 0,Y 183.648,Z 1266.175,A -85,B 0,C 180,E1 2581.028,E2 2581.028} C_VEL
LIN {X 0,Y 189.395,Z 1261.672,A -85,B 0,C 180,E1 2574.881,E2 2574.881} C_VEL
LIN {X 0,Y 197.273,Z 1255.885,A -85,B 0,C 180,E1 2568.797,E2 2568.797} C_VEL
LIN {X 0,Y 207.957,Z 1248.276,A -85,B 0,C 180,E1 2562.653,E2 2562.653} C_VEL
LIN {X 0,Y 223.547,Z 1237.016,A -85,B 0,C 180,E1 2555.961,E2 2555.961} C_VEL
LIN {X 0,Y 236.884,Z 1227.039,A -85,B 0,C 180,E1 2551.517,E2 2551.517} C_VEL
LIN {X 0,Y 250.7,Z 1216.258,A -85,B 0,C 180,E1 2547.716,E2 2547.716} C_VEL
LIN {X 0,Y 265.458,Z 1204.118,A -85,B 0,C 180,E1 2544.303,E2 2544.303} C_VEL
LIN {X 0,Y 285.033,Z 1186.751,A -85,B 0,C 180,E1 2540.531,E2 2540.531} C_VEL
LIN {X 0,Y 300.269,Z 1172.027,A -85,B 0,C 180,E1 2538.041,E2 2538.041} C_VEL
LIN {X 0,Y 314.148,Z 1157.61,A -85,B 0,C 180,E1 2536.036,E2 2536.036} C_VEL
LIN {X 0,Y 328.407,Z 1141.63,A -85,B 0,C 180,E1 2534.197,E2 2534.197} C_VEL
LIN {X 0,Y 345.297,Z 1120.964,A -85,B 0,C 180,E1 2532.264,E2 2532.264} C_VEL
LIN {X 0,Y 360.373,Z 1100.194,A -85,B 0,C 180,E1 2530.714,E2 2530.714} C_VEL
LIN {X 0,Y 372.137,Z 1082.398,A -85,B 0,C 180,E1 2529.612,E2 2529.612} C_VEL
LIN {X 0,Y 383.254,Z 1063.876,A -85,B 0,C 180,E1 2528.634,E2 2528.634} C_VEL
LIN {X 0,Y 394.482,Z 1043.104,A -85,B 0,C 180,E1 2527.718,E2 2527.718} C_VEL
LIN {X 0,Y 406.808,Z 1016.89,A -85,B 0,C 180,E1 2526.776,E2 2526.776} C_VEL
LIN {X 0,Y 415.305,Z 995.878,A -85,B 0,C 180,E1 2526.163,E2 2526.163} C_VEL
LIN {X 0,Y 422.638,Z 974.977,A -85,B 0,C 180,E1 2525.656,E2 2525.656} C_VEL
LIN {X 0,Y 428.94,Z 953.891,A -85,B 0,C 180,E1 2525.232,E2 2525.232} C_VEL
LIN {X 0,Y 434.833,Z 929.993,A -85,B 0,C 180,E1 2524.849,E2 2524.849} C_VEL
LIN {X 0,Y 440.135,Z 900.765,A -85,B 0,C 180,E1 2524.451,E2 2524.451} C_VEL
LIN {X 0,Y 448.281,Z 833.419,A -85,B 0,C 180,E1 2523.593,E2 2523.593} C_VEL
LIN {X 0,Y 458.219,Z 748.923,A -85,B 0,C 180,E1 2522.501,E2 2522.501} C_VEL
LIN {X 0,Y 458.076,Z 746.687,A -85,B 0,C 180,E1 2520.125,E2 2520.125} C_VEL
LIN {X 0,Y 458.044,Z 747.434,A -85,B 0,C 180,E1 2519.124,E2 2519.124} C_VEL
LIN {X 0,Y 458.22,Z 749.112,A -85,B 0,C 180,E1 2517.538,E2 2517.538} C_VEL
LIN {X 0,Y 456.324,Z 765.132,A -85,B 0,C 180,E1 2517.338,E2 2517.338} C_VEL
LIN {X 0,Y 455.366,Z 772.836,A -85,B 0,C 180,E1 2517.367,E2 2517.367} C_VEL
LIN {X 0,Y 452.65,Z 793.482,A -85,B 0,C 180,E1 2517.901,E2 2517.901} C_VEL
LIN {X 0,Y 451.834,Z 800.09,A -85,B 0,C 180,E1 2517.915,E2 2517.915} C_VEL
LIN {X 0,Y 439.721,Z 900.079,A -85,B 0,C 180,E1 2516.672,E2 2516.672} C_VEL
LIN {X 0,Y 434.856,Z 927.778,A -85,B 0,C 180,E1 2516.307,E2 2516.307} C_VEL
LIN {X 0,Y 428.362,Z 954.122,A -85,B 0,C 180,E1 2515.923,E2 2515.923} C_VEL
LIN {X 0,Y 422.175,Z 974.746,A -85,B 0,C 180,E1 2515.552,E2 2515.552} C_VEL
LIN {X 0,Y 414.922,Z 995.389,A -85,B 0,C 180,E1 2515.099,E2 2515.099} C_VEL
LIN {X 0,Y 406.063,Z 1017.224,A -85,B 0,C 180,E1 2514.517,E2 2514.517} C_VEL
LIN {X 0,Y 393.343,Z 1044.094,A -85,B 0,C 180,E1 2513.623,E2 2513.623} C_VEL
LIN {X 0,Y 381.953,Z 1064.965,A -85,B 0,C 180,E1 2512.764,E2 2512.764} C_VEL
LIN {X 0,Y 370.663,Z 1083.587,A -85,B 0,C 180,E1 2511.842,E2 2511.842} C_VEL
LIN {X 0,Y 358.146,Z 1102.3,A -85,B 0,C 180,E1 2510.747,E2 2510.747} C_VEL
LIN {X 0,Y 341.999,Z 1124.151,A -85,B 0,C 180,E1 2509.179,E2 2509.179} C_VEL
LIN {X 0,Y 325.674,Z 1143.771,A -85,B 0,C 180,E1 2507.409,E2 2507.409} C_VEL
LIN {X 0,Y 311.579,Z 1159.348,A -85,B 0,C 180,E1 2505.694,E2 2505.694} C_VEL
LIN {X 0,Y 296.873,Z 1174.39,A -85,B 0,C 180,E1 2503.69,E2 2503.69} C_VEL
LIN {X 0,Y 279.266,Z 1191.097,A -85,B 0,C 180,E1 2500.923,E2 2500.923} C_VEL
LIN {X 0,Y 260.812,Z 1206.989,A -85,B 0,C 180,E1 2497.485,E2 2497.485} C_VEL
LIN {X 0,Y 246.165,Z 1218.789,A -85,B 0,C 180,E1 2494.239,E2 2494.239} C_VEL
LIN {X 0,Y 232.014,Z 1229.596,A -85,B 0,C 180,E1 2490.502,E2 2490.502} C_VEL
LIN {X 0,Y 217.489,Z 1240.202,A -85,B 0,C 180,E1 2485.829,E2 2485.829} C_VEL
LIN {X 0,Y 201.225,Z 1251.576,A -85,B 0,C 180,E1 2479.035,E2 2479.035} C_VEL
LIN {X 0,Y 190.487,Z 1258.998,A -85,B 0,C 180,E1 2473.016,E2 2473.016} C_VEL
LIN {X 0,Y 182.114,Z 1264.953,A -85,B 0,C 180,E1 2466.716,E2 2466.716} C_VEL
LIN {X 0,Y 175.515,Z 1269.988,A -85,B 0,C 180,E1 2459.699,E2 2459.699} C_VEL
LIN {X 0,Y 170.537,Z 1274.539,A -85,B 0,C 180,E1 2450.945,E2 2450.945} C_VEL
LIN {X 0,Y 168.344,Z 1277.277,A -85,B 0,C 180,E1 2442.336,E2 2442.336} C_VEL
LIN {X 0,Y 167.93,Z 1278.477,A -85,B 0,C 180,E1 2435.457,E2 2435.457} C_VEL
LIN {X 0,Y 167.89,Z 1278.797,A -85,B 0,C 180,E1 2429.308,E2 2429.308} C_VEL
LIN {X 0,Y 167.964,Z 1278.37,A -85,B 0,C 180,E1 2423.153,E2 2423.153} C_VEL
LIN {X 0,Y 168.803,Z 1276.52,A -85,B 0,C 180,E1 2414.883,E2 2414.883} C_VEL
LIN {X 0,Y 171.429,Z 1273.528,A -85,B 0,C 180,E1 2406.987,E2 2406.987} C_VEL
LIN {X 0,Y 176.05,Z 1269.522,A -85,B 0,C 180,E1 2399.627,E2 2399.627} C_VEL
LIN {X 0,Y 182.515,Z 1264.617,A -85,B 0,C 180,E1 2392.933,E2 2392.933} C_VEL
LIN {X 0,Y 191.408,Z 1258.312,A -85,B 0,C 180,E1 2386.396,E2 2386.396} C_VEL
LIN {X 0,Y 205.051,Z 1248.897,A -85,B 0,C 180,E1 2379.156,E2 2379.156} C_VEL
LIN {X 0,Y 219.509,Z 1238.63,A -85,B 0,C 180,E1 2373.448,E2 2373.448} C_VEL
LIN {X 0,Y 232.736,Z 1228.953,A -85,B 0,C 180,E1 2369.283,E2 2369.283} C_VEL
LIN {X 0,Y 247.115,Z 1217.932,A -85,B 0,C 180,E1 2365.526,E2 2365.526} C_VEL
LIN {X 0,Y 264.773,Z 1203.627,A -85,B 0,C 180,E1 2361.712,E2 2361.712} C_VEL
LIN {X 0,Y 282.596,Z 1187.788,A -85,B 0,C 180,E1 2358.504,E2 2358.504} C_VEL
LIN {X 0,Y 297.764,Z 1173.305,A -85,B 0,C 180,E1 2356.171,E2 2356.171} C_VEL
LIN {X 0,Y 312.063,Z 1158.615,A -85,B 0,C 180,E1 2354.235,E2 2354.235} C_VEL
LIN {X 0,Y 326.682,Z 1142.381,A -85,B 0,C 180,E1 2352.468,E2 2352.468} C_VEL
LIN {X 0,Y 344.829,Z 1120.141,A -85,B 0,C 180,E1 2350.526,E2 2350.526} C_VEL
LIN {X 0,Y 358.587,Z 1101.318,A -85,B 0,C 180,E1 2349.202,E2 2349.202} C_VEL
LIN {X 0,Y 370.708,Z 1083.131,A -85,B 0,C 180,E1 2348.143,E2 2348.143} C_VEL
LIN {X 0,Y 382.062,Z 1064.352,A -85,B 0,C 180,E1 2347.217,E2 2347.217} C_VEL
LIN {X 0,Y 395.007,Z 1040.481,A -85,B 0,C 180,E1 2346.249,E2 2346.249} C_VEL
LIN {X 0,Y 406.458,Z 1015.698,A -85,B 0,C 180,E1 2345.443,E2 2345.443} C_VEL
LIN {X 0,Y 414.971,Z 994.575,A -85,B 0,C 180,E1 2344.886,E2 2344.886} C_VEL
LIN {X 0,Y 422.225,Z 973.803,A -85,B 0,C 180,E1 2344.433,E2 2344.433} C_VEL
LIN {X 0,Y 429.187,Z 950.246,A -85,B 0,C 180,E1 2344.018,E2 2344.018} C_VEL
LIN {X 0,Y 435.855,Z 921.186,A -85,B 0,C 180,E1 2343.608,E2 2343.608} C_VEL
LIN {X 0,Y 439.748,Z 897.986,A -85,B 0,C 180,E1 2343.304,E2 2343.304} C_VEL
LIN {X 0,Y 456.856,Z 755.792,A -85,B 0,C 180,E1 2341.536,E2 2341.536} C_VEL
LIN {X 0,Y 456.831,Z 754.547,A -85,B 0,C 180,E1 2340.251,E2 2340.251} C_VEL
LIN {X 0,Y 456.827,Z 754.854,A -85,B 0,C 180,E1 2339.122,E2 2339.122} C_VEL
LIN {X 0,Y 456.833,Z 755.921,A -85,B 0,C 180,E1 2338.296,E2 2338.296} C_VEL
LIN {X 0,Y 439.58,Z 898.964,A -85,B 0,C 180,E1 2336.523,E2 2336.523} C_VEL
LIN {X 0,Y 434.87,Z 926.128,A -85,B 0,C 180,E1 2336.168,E2 2336.168} C_VEL
LIN {X 0,Y 428.289,Z 953.009,A -85,B 0,C 180,E1 2335.761,E2 2335.761} C_VEL
LIN {X 0,Y 421.85,Z 974.474,A -85,B 0,C 180,E1 2335.351,E2 2335.351} C_VEL
LIN {X 0,Y 414.62,Z 994.995,A -85,B 0,C 180,E1 2334.876,E2 2334.876} C_VEL
LIN {X 0,Y 405.505,Z 1017.385,A -85,B 0,C 180,E1 2334.25,E2 2334.25} C_VEL
LIN {X 0,Y 393.113,Z 1043.401,A -85,B 0,C 180,E1 2333.348,E2 2333.348} C_VEL
LIN {X 0,Y 381.895,Z 1063.911,A -85,B 0,C 180,E1 2332.478,E2 2332.478} C_VEL
LIN {X 0,Y 370.985,Z 1081.9,A -85,B 0,C 180,E1 2331.563,E2 2331.563} C_VEL
LIN {X 0,Y 358.905,Z 1099.981,A -85,B 0,C 180,E1 2330.49,E2 2330.49} C_VEL
LIN {X 0,Y 344.233,Z 1119.956,A -85,B 0,C 180,E1 2329.058,E2 2329.058} C_VEL
LIN {X 0,Y 326.661,Z 1141.265,A -85,B 0,C 180,E1 2327.149,E2 2327.149} C_VEL
LIN {X 0,Y 312.109,Z 1157.319,A -85,B 0,C 180,E1 2325.364,E2 2325.364} C_VEL
LIN {X 0,Y 298.007,Z 1171.711,A -85,B 0,C 180,E1 2323.429,E2 2323.429} C_VEL
LIN {X 0,Y 282.244,Z 1186.634,A -85,B 0,C 180,E1 2320.978,E2 2320.978} C_VEL
LIN {X 0,Y 262.287,Z 1203.939,A -85,B 0,C 180,E1 2317.311,E2 2317.311} C_VEL
LIN {X 0,Y 247.074,Z 1216.105,A -85,B 0,C 180,E1 2313.96,E2 2313.96} C_VEL
LIN {X 0,Y 233.466,Z 1226.4,A -85,B 0,C 180,E1 2310.4,E2 2310.4} C_VEL
LIN {X 0,Y 220.152,Z 1235.996,A -85,B 0,C 180,E1 2306.226,E2 2306.226} C_VEL
LIN {X 0,Y 205.203,Z 1246.429,A -85,B 0,C 180,E1 2300.333,E2 2300.333} C_VEL
LIN {X 0,Y 192.077,Z 1255.236,A -85,B 0,C 180,E1 2293.414,E2 2293.414} C_VEL
LIN {X 0,Y 183.106,Z 1261.393,A -85,B 0,C 180,E1 2286.928,E2 2286.928} C_VEL
LIN {X 0,Y 176.531,Z 1266.168,A -85,B 0,C 180,E1 2280.281,E2 2280.281} C_VEL
LIN {X 0,Y 171.918,Z 1269.928,A -85,B 0,C 180,E1 2273.228,E2 2273.228} C_VEL
LIN {X 0,Y 169.166,Z 1272.714,A -85,B 0,C 180,E1 2265.786,E2 2265.786} C_VEL
LIN {X 0,Y 168.09,Z 1274.383,A -85,B 0,C 180,E1 2258.562,E2 2258.562} C_VEL
LIN {X 0,Y 167.918,Z 1275.008,A -85,B 0,C 180,E1 2252.399,E2 2252.399} C_VEL
LIN {X 0,Y 167.923,Z 1274.975,A -85,B 0,C 180,E1 2246.938,E2 2246.938} C_VEL
LIN {X 0,Y 168.111,Z 1274.35,A -85,B 0,C 180,E1 2241.114,E2 2241.114} C_VEL
LIN {X 0,Y 169.229,Z 1272.658,A -85,B 0,C 180,E1 2233.888,E2 2233.888} C_VEL
LIN {X 0,Y 171.903,Z 1269.971,A -85,B 0,C 180,E1 2226.713,E2 2226.713} C_VEL
LIN {X 0,Y 176.452,Z 1266.265,A -85,B 0,C 180,E1 2219.726,E2 2219.726} C_VEL
LIN {X 0,Y 183.005,Z 1261.511,A -85,B 0,C 180,E1 2213.071,E2 2213.071} C_VEL
LIN {X 0,Y 191.957,Z 1255.376,A -85,B 0,C 180,E1 2206.576,E2 2206.576} C_VEL
LIN {X 0,Y 205.09,Z 1246.596,A -85,B 0,C 180,E1 2199.634,E2 2199.634} C_VEL
LIN {X 0,Y 220,Z 1236.196,A -85,B 0,C 180,E1 2193.741,E2 2193.741} C_VEL
LIN {X 0,Y 233.538,Z 1226.45,A -85,B 0,C 180,E1 2189.497,E2 2189.497} C_VEL
LIN {X 0,Y 247.657,Z 1215.778,A -85,B 0,C 180,E1 2185.818,E2 2185.818} C_VEL
LIN {X 0,Y 265.276,Z 1201.684,A -85,B 0,C 180,E1 2182.016,E2 2182.016} C_VEL
LIN {X 0,Y 283.586,Z 1185.565,A -85,B 0,C 180,E1 2178.715,E2 2178.715} C_VEL
LIN {X 0,Y 298.157,Z 1171.764,A -85,B 0,C 180,E1 2176.468,E2 2176.468} C_VEL
LIN {X 0,Y 312.837,Z 1156.776,A -85,B 0,C 180,E1 2174.463,E2 2174.463} C_VEL
LIN {X 0,Y 328.316,Z 1139.646,A -85,B 0,C 180,E1 2172.585,E2 2172.585} C_VEL
LIN {X 0,Y 345.92,Z 1118.019,A -85,B 0,C 180,E1 2170.69,E2 2170.69} C_VEL
LIN {X 0,Y 359.333,Z 1099.713,A -85,B 0,C 180,E1 2169.391,E2 2169.391} C_VEL
LIN {X 0,Y 371.329,Z 1081.75,A -85,B 0,C 180,E1 2168.329,E2 2168.329} C_VEL
LIN {X 0,Y 382.588,Z 1063.151,A -85,B 0,C 180,E1 2167.389,E2 2167.389} C_VEL
LIN {X 0,Y 395.378,Z 1039.593,A -85,B 0,C 180,E1 2166.407,E2 2166.407} C_VEL
LIN {X 0,Y 406.833,Z 1014.85,A -85,B 0,C 180,E1 2165.579,E2 2165.579} C_VEL
LIN {X 0,Y 414.998,Z 994.676,A -85,B 0,C 180,E1 2165.022,E2 2165.022} C_VEL
LIN {X 0,Y 422.233,Z 974.098,A -85,B 0,C 180,E1 2164.547,E2 2164.547} C_VEL
LIN {X 0,Y 428.752,Z 952.287,A -85,B 0,C 180,E1 2164.132,E2 2164.132} C_VEL
LIN {X 0,Y 435.413,Z 924.637,A -85,B 0,C 180,E1 2163.72,E2 2163.72} C_VEL
LIN {X 0,Y 439.891,Z 898.649,A -85,B 0,C 180,E1 2163.38,E2 2163.38} C_VEL
LIN {X 0,Y 457.09,Z 756.074,A -85,B 0,C 180,E1 2161.601,E2 2161.601} C_VEL
LIN {X 0,Y 457.1,Z 754.631,A -85,B 0,C 180,E1 2160,E2 2160} C_VEL
LIN {X 0,Y 457.065,Z 756.373,A -85,B 0,C 180,E1 2158.453,E2 2158.453} C_VEL
LIN {X 0,Y 451.834,Z 800.09,A -85,B 0,C 180,E1 2157.915,E2 2157.915} C_VEL
LIN {X 0,Y 450.879,Z 807.791,A -85,B 0,C 180,E1 2157.945,E2 2157.945} C_VEL
LIN {X 0,Y 448.206,Z 828.429,A -85,B 0,C 180,E1 2158.491,E2 2158.491} C_VEL
LIN {X 0,Y 447.39,Z 835.039,A -85,B 0,C 180,E1 2158.512,E2 2158.512} C_VEL
LIN {X 0,Y 439.13,Z 901.406,A -85,B 0,C 180,E1 2157.701,E2 2157.701} C_VEL
LIN {X 0,Y 433.627,Z 931.044,A -85,B 0,C 180,E1 2157.32,E2 2157.32} C_VEL
LIN {X 0,Y 427.651,Z 954.804,A -85,B 0,C 180,E1 2156.986,E2 2156.986} C_VEL
LIN {X 0,Y 421.382,Z 975.409,A -85,B 0,C 180,E1 2156.63,E2 2156.63} C_VEL
LIN {X 0,Y 413.823,Z 996.595,A -85,B 0,C 180,E1 2156.183,E2 2156.183} C_VEL
LIN {X 0,Y 403.629,Z 1021.213,A -85,B 0,C 180,E1 2155.541,E2 2155.541} C_VEL
LIN {X 0,Y 391.343,Z 1046.221,A -85,B 0,C 180,E1 2154.722,E2 2154.722} C_VEL
LIN {X 0,Y 380.581,Z 1065.613,A -85,B 0,C 180,E1 2153.95,E2 2153.95} C_VEL
LIN {X 0,Y 369.59,Z 1083.502,A -85,B 0,C 180,E1 2153.099,E2 2153.099} C_VEL
LIN {X 0,Y 356.851,Z 1102.31,A -85,B 0,C 180,E1 2152.043,E2 2152.043} C_VEL
LIN {X 0,Y 340.469,Z 1124.158,A -85,B 0,C 180,E1 2150.534,E2 2150.534} C_VEL
LIN {X 0,Y 324.041,Z 1143.603,A -85,B 0,C 180,E1 2148.846,E2 2148.846} C_VEL
LIN {X 0,Y 310.047,Z 1158.824,A -85,B 0,C 180,E1 2147.237,E2 2147.237} C_VEL
LIN {X 0,Y 295.508,Z 1173.453,A -85,B 0,C 180,E1 2145.369,E2 2145.369} C_VEL
LIN {X 0,Y 280.015,Z 1187.91,A -85,B 0,C 180,E1 2143.104,E2 2143.104} C_VEL
LIN {X 0,Y 260.125,Z 1204.983,A -85,B 0,C 180,E1 2139.677,E2 2139.677} C_VEL
LIN {X 0,Y 243.572,Z 1217.985,A -85,B 0,C 180,E1 2136.245,E2 2136.245} C_VEL
LIN {X 0,Y 228.698,Z 1228.987,A -85,B 0,C 180,E1 2132.544,E2 2132.544} C_VEL
LIN {X 0,Y 214.182,Z 1239.186,A -85,B 0,C 180,E1 2128.155,E2 2128.155} C_VEL
LIN {X 0,Y 198.076,Z 1250.058,A -85,B 0,C 180,E1 2121.934,E2 2121.934} C_VEL
LIN {X 0,Y 184.923,Z 1258.601,A -85,B 0,C 180,E1 2115.083,E2 2115.083} C_VEL
LIN {X 0,Y 175.902,Z 1264.585,A -85,B 0,C 180,E1 2108.688,E2 2108.688} C_VEL
LIN {X 0,Y 168.927,Z 1269.479,A -85,B 0,C 180,E1 2101.776,E2 2101.776} C_VEL
LIN {X 0,Y 163.858,Z 1273.475,A -85,B 0,C 180,E1 2094.12,E2 2094.12} C_VEL
LIN {X 0,Y 160.938,Z 1276.457,A -85,B 0,C 180,E1 2085.853,E2 2085.853} C_VEL
LIN {X 0,Y 159.984,Z 1278.234,A -85,B 0,C 180,E1 2077.531,E2 2077.531} C_VEL
LIN {X 0,Y 159.893,Z 1278.691,A -85,B 0,C 180,E1 2071.065,E2 2071.065} C_VEL
LIN {X 0,Y 159.924,Z 1278.431,A -85,B 0,C 180,E1 2064.968,E2 2064.968} C_VEL
LIN {X 0,Y 160.184,Z 1277.521,A -85,B 0,C 180,E1 2058.833,E2 2058.833} C_VEL
LIN {X 0,Y 161.378,Z 1275.851,A -85,B 0,C 180,E1 2052.316,E2 2052.316} C_VEL
LIN {X 0,Y 164.252,Z 1273.09,A -85,B 0,C 180,E1 2045.1,E2 2045.1} C_VEL
LIN {X 0,Y 169.226,Z 1269.221,A -85,B 0,C 180,E1 2037.865,E2 2037.865} C_VEL
LIN {X 0,Y 176.7,Z 1264.01,A -85,B 0,C 180,E1 2030.661,E2 2030.661} C_VEL
LIN {X 0,Y 188.893,Z 1256.035,A -85,B 0,C 180,E1 2022.616,E2 2022.616} C_VEL
LIN {X 0,Y 202.83,Z 1246.76,A -85,B 0,C 180,E1 2016.043,E2 2016.043} C_VEL
LIN {X 0,Y 216.201,Z 1237.684,A -85,B 0,C 180,E1 2011.165,E2 2011.165} C_VEL
LIN {X 0,Y 230.173,Z 1227.822,A -85,B 0,C 180,E1 2007.049,E2 2007.049} C_VEL
LIN {X 0,Y 248.252,Z 1214.374,A -85,B 0,C 180,E1 2002.718,E2 2002.718} C_VEL
LIN {X 0,Y 266.688,Z 1199.33,A -85,B 0,C 180,E1 1999.112,E2 1999.112} C_VEL
LIN {X 0,Y 281.754,Z 1186.145,A -85,B 0,C 180,E1 1996.618,E2 1996.618} C_VEL
LIN {X 0,Y 296.921,Z 1171.877,A -85,B 0,C 180,E1 1994.43,E2 1994.43} C_VEL
LIN {X 0,Y 313.495,Z 1155.013,A -85,B 0,C 180,E1 1992.339,E2 1992.339} C_VEL
LIN {X 0,Y 332.297,Z 1133.756,A -85,B 0,C 180,E1 1990.266,E2 1990.266} C_VEL
LIN {X 0,Y 346.156,Z 1116.448,A -85,B 0,C 180,E1 1988.915,E2 1988.915} C_VEL
LIN {X 0,Y 358.802,Z 1099.178,A -85,B 0,C 180,E1 1987.78,E2 1987.78} C_VEL
LIN {X 0,Y 371.533,Z 1080.09,A -85,B 0,C 180,E1 1986.734,E2 1986.734} C_VEL
LIN {X 0,Y 385.971,Z 1055.84,A -85,B 0,C 180,E1 1985.649,E2 1985.649} C_VEL
LIN {X 0,Y 397.39,Z 1033.762,A -85,B 0,C 180,E1 1984.853,E2 1984.853} C_VEL
LIN {X 0,Y 406.632,Z 1013.587,A -85,B 0,C 180,E1 1984.249,E2 1984.249} C_VEL
LIN {X 0,Y 414.848,Z 993.192,A -85,B 0,C 180,E1 1983.743,E2 1983.743} C_VEL
LIN {X 0,Y 422.656,Z 970.743,A -85,B 0,C 180,E1 1983.286,E2 1983.286} C_VEL
LIN {X 0,Y 430.859,Z 941.679,A -85,B 0,C 180,E1 1982.824,E2 1982.824} C_VEL
LIN {X 0,Y 435.982,Z 918.107,A -85,B 0,C 180,E1 1982.515,E2 1982.515} C_VEL
LIN {X 0,Y 439.657,Z 895.773,A -85,B 0,C 180,E1 1982.231,E2 1982.231} C_VEL
LIN {X 0,Y 455.846,Z 762.776,A -85,B 0,C 180,E1 1980.597,E2 1980.597} C_VEL
LIN {X 0,Y 455.854,Z 762.593,A -85,B 0,C 180,E1 1979.372,E2 1979.372} C_VEL
LIN {X 0,Y 455.822,Z 762.965,A -85,B 0,C 180,E1 1979.219,E2 1979.219} C_VEL
LIN {X 0,Y 439.167,Z 899.073,A -85,B 0,C 180,E1 1977.568,E2 1977.568} C_VEL
LIN {X 0,Y 434.377,Z 926.382,A -85,B 0,C 180,E1 1977.221,E2 1977.221} C_VEL
LIN {X 0,Y 427.739,Z 953.217,A -85,B 0,C 180,E1 1976.832,E2 1976.832} C_VEL
LIN {X 0,Y 421.274,Z 974.57,A -85,B 0,C 180,E1 1976.442,E2 1976.442} C_VEL
LIN {X 0,Y 413.902,Z 995.293,A -85,B 0,C 180,E1 1975.983,E2 1975.983} C_VEL
LIN {X 0,Y 404.775,Z 1017.48,A -85,B 0,C 180,E1 1975.388,E2 1975.388} C_VEL
LIN {X 0,Y 392.256,Z 1043.496,A -85,B 0,C 180,E1 1974.525,E2 1974.525} C_VEL
LIN {X 0,Y 380.781,Z 1064.232,A -85,B 0,C 180,E1 1973.681,E2 1973.681} C_VEL
LIN {X 0,Y 369.403,Z 1082.726,A -85,B 0,C 180,E1 1972.775,E2 1972.775} C_VEL
LIN {X 0,Y 357.176,Z 1100.741,A -85,B 0,C 180,E1 1971.742,E2 1971.742} C_VEL
LIN {X 0,Y 340.925,Z 1122.434,A -85,B 0,C 180,E1 1970.225,E2 1970.225} C_VEL
LIN {X 0,Y 324.02,Z 1142.368,A -85,B 0,C 180,E1 1968.468,E2 1968.468} C_VEL
LIN {X 0,Y 310.122,Z 1157.413,A -85,B 0,C 180,E1 1966.843,E2 1966.843} C_VEL
LIN {X 0,Y 296.051,Z 1171.507,A -85,B 0,C 180,E1 1965.015,E2 1965.015} C_VEL
LIN {X 0,Y 280.609,Z 1185.844,A -85,B 0,C 180,E1 1962.749,E2 1962.749} C_VEL
LIN {X 0,Y 261.598,Z 1202.14,A -85,B 0,C 180,E1 1959.474,E2 1959.474} C_VEL
LIN {X 0,Y 243.735,Z 1216.036,A -85,B 0,C 180,E1 1955.78,E2 1955.78} C_VEL
LIN {X 0,Y 229.345,Z 1226.562,A -85,B 0,C 180,E1 1952.193,E2 1952.193} C_VEL
LIN {X 0,Y 215.605,Z 1236.089,A -85,B 0,C 180,E1 1948.079,E2 1948.079} C_VEL
LIN {X 0,Y 199.981,Z 1246.504,A -85,B 0,C 180,E1 1942.194,E2 1942.194} C_VEL
LIN {X 0,Y 186.097,Z 1255.328,A -85,B 0,C 180,E1 1935.182,E2 1935.182} C_VEL
LIN {X 0,Y 176.522,Z 1261.485,A -85,B 0,C 180,E1 1928.551,E2 1928.551} C_VEL
LIN {X 0,Y 169.439,Z 1266.259,A -85,B 0,C 180,E1 1921.692,E2 1921.692} C_VEL
LIN {X 0,Y 164.218,Z 1270.164,A -85,B 0,C 180,E1 1914.031,E2 1914.031} C_VEL
LIN {X 0,Y 161.075,Z 1273.138,A -85,B 0,C 180,E1 1905.491,E2 1905.491} C_VEL
LIN {X 0,Y 160.02,Z 1274.833,A -85,B 0,C 180,E1 1896.828,E2 1896.828} C_VEL
LIN {X 0,Y 159.908,Z 1275.251,A -85,B 0,C 180,E1 1890.01,E2 1890.01} C_VEL
LIN {X 0,Y 160.016,Z 1274.844,A -85,B 0,C 180,E1 1883.192,E2 1883.192} C_VEL
LIN {X 0,Y 161.052,Z 1273.193,A -85,B 0,C 180,E1 1874.528,E2 1874.528} C_VEL
LIN {X 0,Y 164.191,Z 1270.217,A -85,B 0,C 180,E1 1865.932,E2 1865.932} C_VEL
LIN {X 0,Y 169.356,Z 1266.354,A -85,B 0,C 180,E1 1858.314,E2 1858.314} C_VEL
LIN {X 0,Y 176.42,Z 1261.601,A -85,B 0,C 180,E1 1851.446,E2 1851.446} C_VEL
LIN {X 0,Y 185.493,Z 1255.766,A -85,B 0,C 180,E1 1845.093,E2 1845.093} C_VEL
LIN {X 0,Y 198.688,Z 1247.408,A -85,B 0,C 180,E1 1838.29,E2 1838.29} C_VEL
LIN {X 0,Y 214.794,Z 1236.741,A -85,B 0,C 180,E1 1832.107,E2 1832.107} C_VEL
LIN {X 0,Y 229.29,Z 1226.708,A -85,B 0,C 180,E1 1827.739,E2 1827.739} C_VEL
LIN {X 0,Y 244.125,Z 1215.868,A -85,B 0,C 180,E1 1824.048,E2 1824.048} C_VEL
LIN {X 0,Y 262.445,Z 1201.625,A -85,B 0,C 180,E1 1820.286,E2 1820.286} C_VEL
LIN {X 0,Y 281.306,Z 1185.396,A -85,B 0,C 180,E1 1817.06,E2 1817.06} C_VEL
LIN {X 0,Y 296.411,Z 1171.365,A -85,B 0,C 180,E1 1814.855,E2 1814.855} C_VEL
LIN {X 0,Y 310.874,Z 1156.863,A -85,B 0,C 180,E1 1812.986,E2 1812.986} C_VEL
LIN {X 0,Y 326.612,Z 1139.741,A -85,B 0,C 180,E1 1811.174,E2 1811.174} C_VEL
LIN {X 0,Y 344.491,Z 1118.104,A -85,B 0,C 180,E1 1809.348,E2 1809.348} C_VEL
LIN {X 0,Y 357.992,Z 1099.935,A -85,B 0,C 180,E1 1808.106,E2 1808.106} C_VEL
LIN {X 0,Y 370.166,Z 1081.941,A -85,B 0,C 180,E1 1807.084,E2 1807.084} C_VEL
LIN {X 0,Y 381.15,Z 1064.044,A -85,B 0,C 180,E1 1806.213,E2 1806.213} C_VEL
LIN {X 0,Y 392.632,Z 1043.271,A -85,B 0,C 180,E1 1805.37,E2 1805.37} C_VEL
LIN {X 0,Y 405.421,Z 1016.579,A -85,B 0,C 180,E1 1804.491,E2 1804.491} C_VEL
LIN {X 0,Y 414.37,Z 994.756,A -85,B 0,C 180,E1 1803.91,E2 1803.91} C_VEL
LIN {X 0,Y 421.671,Z 974.177,A -85,B 0,C 180,E1 1803.456,E2 1803.456} C_VEL
LIN {X 0,Y 428.278,Z 952.258,A -85,B 0,C 180,E1 1803.058,E2 1803.058} C_VEL
LIN {X 0,Y 435.027,Z 924.384,A -85,B 0,C 180,E1 1802.661,E2 1802.661} C_VEL
LIN {X 0,Y 439.491,Z 898.716,A -85,B 0,C 180,E1 1802.336,E2 1802.336} C_VEL
LIN {X 0,Y 456.086,Z 763.107,A -85,B 0,C 180,E1 1800.667,E2 1800.667} C_VEL
LIN {X 0,Y 456.12,Z 762.63,A -85,B 0,C 180,E1 1799.874,E2 1799.874} C_VEL
LIN {X 0,Y 456.066,Z 763.312,A -85,B 0,C 180,E1 1799.377,E2 1799.377} C_VEL
LIN {X 0,Y 447.39,Z 835.039,A -85,B 0,C 180,E1 1798.512,E2 1798.512} C_VEL
LIN {X 0,Y 446.435,Z 842.745,A -85,B 0,C 180,E1 1798.551,E2 1798.551} C_VEL
LIN {X 0,Y 443.808,Z 863.38,A -85,B 0,C 180,E1 1799.108,E2 1799.108} C_VEL
LIN {X 0,Y 442.995,Z 869.985,A -85,B 0,C 180,E1 1799.124,E2 1799.124} C_VEL
LIN {X 0,Y 437.771,Z 908.584,A -85,B 0,C 180,E1 1798.661,E2 1798.661} C_VEL
LIN {X 0,Y 432.429,Z 934.752,A -85,B 0,C 180,E1 1798.334,E2 1798.334} C_VEL
LIN {X 0,Y 426.788,Z 956.541,A -85,B 0,C 180,E1 1798.037,E2 1798.037} C_VEL
LIN {X 0,Y 420.177,Z 977.761,A -85,B 0,C 180,E1 1797.681,E2 1797.681} C_VEL
LIN {X 0,Y 410.912,Z 1002.945,A -85,B 0,C 180,E1 1797.155,E2 1797.155} C_VEL
LIN {X 0,Y 399.66,Z 1028.273,A -85,B 0,C 180,E1 1796.484,E2 1796.484} C_VEL
LIN {X 0,Y 389.441,Z 1048.438,A -85,B 0,C 180,E1 1795.829,E2 1795.829} C_VEL
LIN {X 0,Y 378.794,Z 1067.237,A -85,B 0,C 180,E1 1795.102,E2 1795.102} C_VEL
LIN {X 0,Y 366.351,Z 1087.027,A -85,B 0,C 180,E1 1794.182,E2 1794.182} C_VEL
LIN {X 0,Y 349.173,Z 1111.242,A -85,B 0,C 180,E1 1792.795,E2 1792.795} C_VEL
LIN {X 0,Y 334.605,Z 1129.545,A -85,B 0,C 180,E1 1791.487,E2 1791.487} C_VEL
LIN {X 0,Y 320.237,Z 1146.059,A -85,B 0,C 180,E1 1790.051,E2 1790.051} C_VEL
LIN {X 0,Y 305.182,Z 1161.956,A -85,B 0,C 180,E1 1788.376,E2 1788.376} C_VEL
LIN {X 0,Y 285.566,Z 1180.853,A -85,B 0,C 180,E1 1785.871,E2 1785.871} C_VEL
LIN {X 0,Y 268.261,Z 1195.911,A -85,B 0,C 180,E1 1783.288,E2 1783.288} C_VEL
LIN {X 0,Y 252.813,Z 1208.393,A -85,B 0,C 180,E1 1780.596,E2 1780.596} C_VEL
LIN {X 0,Y 237.165,Z 1220.204,A -85,B 0,C 180,E1 1777.389,E2 1777.389} C_VEL
LIN {X 0,Y 219.003,Z 1233.095,A -85,B 0,C 180,E1 1772.834,E2 1772.834} C_VEL
LIN {X 0,Y 201.512,Z 1244.503,A -85,B 0,C 180,E1 1767.258,E2 1767.258} C_VEL
LIN {X 0,Y 188.286,Z 1252.822,A -85,B 0,C 180,E1 1761.791,E2 1761.791} C_VEL
LIN {X 0,Y 176.613,Z 1260.043,A -85,B 0,C 180,E1 1755.492,E2 1755.492} C_VEL
LIN {X 0,Y 165.223,Z 1267.291,A -85,B 0,C 180,E1 1746.793,E2 1746.793} C_VEL
LIN {X 0,Y 157.636,Z 1272.41,A -85,B 0,C 180,E1 1737.57,E2 1737.57} C_VEL
LIN {X 0,Y 153.942,Z 1275.44,A -85,B 0,C 180,E1 1729.728,E2 1729.728} C_VEL
LIN {X 0,Y 152.345,Z 1277.31,A -85,B 0,C 180,E1 1722.497,E2 1722.497} C_VEL
LIN {X 0,Y 151.934,Z 1278.325,A -85,B 0,C 180,E1 1715.654,E2 1715.654} C_VEL
LIN {X 0,Y 151.891,Z 1278.622,A -85,B 0,C 180,E1 1709.235,E2 1709.235} C_VEL
LIN {X 0,Y 151.985,Z 1278.193,A -85,B 0,C 180,E1 1702.429,E2 1702.429} C_VEL
LIN {X 0,Y 153.019,Z 1276.457,A -85,B 0,C 180,E1 1693.671,E2 1693.671} C_VEL
LIN {X 0,Y 156.177,Z 1273.509,A -85,B 0,C 180,E1 1684.994,E2 1684.994} C_VEL
LIN {X 0,Y 161.625,Z 1269.549,A -85,B 0,C 180,E1 1677.005,E2 1677.005} C_VEL
LIN {X 0,Y 169.48,Z 1264.433,A -85,B 0,C 180,E1 1669.525,E2 1669.525} C_VEL
LIN {X 0,Y 179.632,Z 1258.126,A -85,B 0,C 180,E1 1662.703,E2 1662.703} C_VEL
LIN {X 0,Y 194.873,Z 1248.71,A -85,B 0,C 180,E1 1655.32,E2 1655.32} C_VEL
LIN {X 0,Y 210.574,Z 1238.515,A -85,B 0,C 180,E1 1649.652,E2 1649.652} C_VEL
LIN {X 0,Y 224.972,Z 1228.765,A -85,B 0,C 180,E1 1645.535,E2 1645.535} C_VEL
LIN {X 0,Y 240.344,Z 1217.744,A -85,B 0,C 180,E1 1641.904,E2 1641.904} C_VEL
LIN {X 0,Y 259.87,Z 1202.759,A -85,B 0,C 180,E1 1638.115,E2 1638.115} C_VEL
LIN {X 0,Y 278.61,Z 1186.825,A -85,B 0,C 180,E1 1635.104,E2 1635.104} C_VEL
LIN {X 0,Y 294.159,Z 1172.542,A -85,B 0,C 180,E1 1632.964,E2 1632.964} C_VEL
LIN {X 0,Y 309.755,Z 1157.032,A -85,B 0,C 180,E1 1631.081,E2 1631.081} C_VEL
LIN {X 0,Y 328.14,Z 1137.006,A -85,B 0,C 180,E1 1629.136,E2 1629.136} C_VEL
LIN {X 0,Y 344.034,Z 1117.575,A -85,B 0,C 180,E1 1627.647,E2 1627.647} C_VEL
LIN {X 0,Y 356.806,Z 1100.46,A -85,B 0,C 180,E1 1626.557,E2 1626.557} C_VEL
LIN {X 0,Y 369.066,Z 1082.448,A -85,B 0,C 180,E1 1625.597,E2 1625.597} C_VEL
LIN {X 0,Y 380.896,Z 1063.255,A -85,B 0,C 180,E1 1624.739,E2 1624.739} C_VEL
LIN {X 0,Y 394.353,Z 1038.702,A -85,B 0,C 180,E1 1623.844,E2 1623.844} C_VEL
LIN {X 0,Y 405.574,Z 1014.737,A -85,B 0,C 180,E1 1623.142,E2 1623.142} C_VEL
LIN {X 0,Y 413.908,Z 994.383,A -85,B 0,C 180,E1 1622.657,E2 1622.657} C_VEL
LIN {X 0,Y 421.286,Z 973.608,A -85,B 0,C 180,E1 1622.247,E2 1622.247} C_VEL
LIN {X 0,Y 428.256,Z 950.415,A -85,B 0,C 180,E1 1621.876,E2 1621.876} C_VEL
LIN {X 0,Y 435.108,Z 921.141,A -85,B 0,C 180,E1 1621.497,E2 1621.497} C_VEL
LIN {X 0,Y 439.102,Z 897.855,A -85,B 0,C 180,E1 1621.21,E2 1621.21} C_VEL
LIN {X 0,Y 452.52,Z 789.592,A -85,B 0,C 180,E1 1619.915,E2 1619.915} C_VEL
LIN {X 0,Y 438.854,Z 899.503,A -85,B 0,C 180,E1 1618.61,E2 1618.61} C_VEL
LIN {X 0,Y 433.932,Z 927.069,A -85,B 0,C 180,E1 1618.271,E2 1618.271} C_VEL
LIN {X 0,Y 427.309,Z 953.532,A -85,B 0,C 180,E1 1617.904,E2 1617.904} C_VEL
LIN {X 0,Y 420.851,Z 974.667,A -85,B 0,C 180,E1 1617.536,E2 1617.536} C_VEL
LIN {X 0,Y 413.492,Z 995.188,A -85,B 0,C 180,E1 1617.102,E2 1617.102} C_VEL
LIN {X 0,Y 404.205,Z 1017.576,A -85,B 0,C 180,E1 1616.53,E2 1616.53} C_VEL
LIN {X 0,Y 391.565,Z 1043.59,A -85,B 0,C 180,E1 1615.707,E2 1615.707} C_VEL
LIN {X 0,Y 379.973,Z 1064.326,A -85,B 0,C 180,E1 1614.9,E2 1614.9} C_VEL
LIN {X 0,Y 368.466,Z 1082.82,A -85,B 0,C 180,E1 1614.034,E2 1614.034} C_VEL
LIN {X 0,Y 355.619,Z 1101.5,A -85,B 0,C 180,E1 1613.006,E2 1613.006} C_VEL
LIN {X 0,Y 338.691,Z 1123.633,A -85,B 0,C 180,E1 1611.506,E2 1611.506} C_VEL
LIN {X 0,Y 322.48,Z 1142.453,A -85,B 0,C 180,E1 1609.904,E2 1609.904} C_VEL
LIN {X 0,Y 308.344,Z 1157.507,A -85,B 0,C 180,E1 1608.34,E2 1608.34} C_VEL
LIN {X 0,Y 294.013,Z 1171.601,A -85,B 0,C 180,E1 1606.579,E2 1606.579} C_VEL
LIN {X 0,Y 278.007,Z 1186.156,A -85,B 0,C 180,E1 1604.351,E2 1604.351} C_VEL
LIN {X 0,Y 257.958,Z 1202.865,A -85,B 0,C 180,E1 1601.059,E2 1601.059} C_VEL
LIN {X 0,Y 240.983,Z 1215.723,A -85,B 0,C 180,E1 1597.721,E2 1597.721} C_VEL
LIN {X 0,Y 225.656,Z 1226.587,A -85,B 0,C 180,E1 1594.103,E2 1594.103} C_VEL
LIN {X 0,Y 211.287,Z 1236.183,A -85,B 0,C 180,E1 1590.011,E2 1590.011} C_VEL
LIN {X 0,Y 194.959,Z 1246.597,A -85,B 0,C 180,E1 1584.139,E2 1584.139} C_VEL
LIN {X 0,Y 180.033,Z 1255.58,A -85,B 0,C 180,E1 1576.911,E2 1576.911} C_VEL
LIN {X 0,Y 170.091,Z 1261.577,A -85,B 0,C 180,E1 1570.299,E2 1570.299} C_VEL
LIN {X 0,Y 162.342,Z 1266.42,A -85,B 0,C 180,E1 1563.107,E2 1563.107} C_VEL
LIN {X 0,Y 156.549,Z 1270.402,A -85,B 0,C 180,E1 1554.91,E2 1554.91} C_VEL
LIN {X 0,Y 152.983,Z 1273.558,A -85,B 0,C 180,E1 1545.166,E2 1545.166} C_VEL
LIN {X 0,Y 152.002,Z 1274.964,A -85,B 0,C 180,E1 1536.431,E2 1536.431} C_VEL
LIN {X 0,Y 151.897,Z 1275.329,A -85,B 0,C 180,E1 1529.634,E2 1529.634} C_VEL
LIN {X 0,Y 152.033,Z 1274.932,A -85,B 0,C 180,E1 1522.833,E2 1522.833} C_VEL
LIN {X 0,Y 153.217,Z 1273.281,A -85,B 0,C 180,E1 1513.715,E2 1513.715} C_VEL
LIN {X 0,Y 156.71,Z 1270.307,A -85,B 0,C 180,E1 1504.704,E2 1504.704} C_VEL
LIN {X 0,Y 162.369,Z 1266.444,A -85,B 0,C 180,E1 1496.779,E2 1496.779} C_VEL
LIN {X 0,Y 169.986,Z 1261.691,A -85,B 0,C 180,E1 1489.696,E2 1489.696} C_VEL
LIN {X 0,Y 180.182,Z 1255.557,A -85,B 0,C 180,E1 1482.919,E2 1482.919} C_VEL
LIN {X 0,Y 194.94,Z 1246.699,A -85,B 0,C 180,E1 1475.784,E2 1475.784} C_VEL
LIN {X 0,Y 211.141,Z 1236.376,A -85,B 0,C 180,E1 1469.952,E2 1469.952} C_VEL
LIN {X 0,Y 225.507,Z 1226.798,A -85,B 0,C 180,E1 1465.852,E2 1465.852} C_VEL
LIN {X 0,Y 240.833,Z 1215.958,A -85,B 0,C 180,E1 1462.228,E2 1462.228} C_VEL
LIN {X 0,Y 259.469,Z 1201.862,A -85,B 0,C 180,E1 1458.589,E2 1458.589} C_VEL
LIN {X 0,Y 278.112,Z 1186.251,A -85,B 0,C 180,E1 1455.553,E2 1455.553} C_VEL
LIN {X 0,Y 293.877,Z 1171.94,A -85,B 0,C 180,E1 1453.359,E2 1453.359} C_VEL
LIN {X 0,Y 309.119,Z 1156.951,A -85,B 0,C 180,E1 1451.491,E2 1451.491} C_VEL
LIN {X 0,Y 325.263,Z 1139.666,A -85,B 0,C 180,E1 1449.734,E2 1449.734} C_VEL
LIN {X 0,Y 343.642,Z 1117.688,A -85,B 0,C 180,E1 1447.961,E2 1447.961} C_VEL
LIN {X 0,Y 357.403,Z 1099.354,A -85,B 0,C 180,E1 1446.765,E2 1446.765} C_VEL
LIN {X 0,Y 369.795,Z 1081.186,A -85,B 0,C 180,E1 1445.784,E2 1445.784} C_VEL
LIN {X 0,Y 381.801,Z 1061.699,A -85,B 0,C 180,E1 1444.892,E2 1444.892} C_VEL
LIN {X 0,Y 395.839,Z 1035.787,A -85,B 0,C 180,E1 1443.931,E2 1443.931} C_VEL
LIN {X 0,Y 406.069,Z 1013.884,A -85,B 0,C 180,E1 1443.274,E2 1443.274} C_VEL
LIN {X 0,Y 414.402,Z 993.518,A -85,B 0,C 180,E1 1442.766,E2 1442.766} C_VEL
LIN {X 0,Y 421.755,Z 972.776,A -85,B 0,C 180,E1 1442.335,E2 1442.335} C_VEL
LIN {X 0,Y 429.36,Z 947.295,A -85,B 0,C 180,E1 1441.908,E2 1441.908} C_VEL
LIN {X 0,Y 435.623,Z 919.752,A -85,B 0,C 180,E1 1441.546,E2 1441.546} C_VEL
LIN {X 0,Y 439.475,Z 897.132,A -85,B 0,C 180,E1 1441.27,E2 1441.27} C_VEL
LIN {X 0,Y 452.357,Z 793.259,A -85,B 0,C 180,E1 1440.033,E2 1440.033} C_VEL
LIN {X 0,Y 442.995,Z 869.985,A -85,B 0,C 180,E1 1439.124,E2 1439.124} C_VEL
LIN {X 0,Y 442.065,Z 877.684,A -85,B 0,C 180,E1 1439.166,E2 1439.166} C_VEL
LIN {X 0,Y 439.235,Z 898.279,A -85,B 0,C 180,E1 1439.739,E2 1439.739} C_VEL
LIN {X 0,Y 438.256,Z 904.869,A -85,B 0,C 180,E1 1439.756,E2 1439.756} C_VEL
LIN {X 0,Y 432.643,Z 933.112,A -85,B 0,C 180,E1 1439.418,E2 1439.418} C_VEL
LIN {X 0,Y 426.87,Z 955.479,A -85,B 0,C 180,E1 1439.13,E2 1439.13} C_VEL
LIN {X 0,Y 420.339,Z 976.456,A -85,B 0,C 180,E1 1438.801,E2 1438.801} C_VEL
LIN {X 0,Y 412.568,Z 997.72,A -85,B 0,C 180,E1 1438.392,E2 1438.392} C_VEL
LIN {X 0,Y 401.215,Z 1024.165,A -85,B 0,C 180,E1 1437.757,E2 1437.757} C_VEL
LIN {X 0,Y 389.865,Z 1046.641,A -85,B 0,C 180,E1 1437.082,E2 1437.082} C_VEL
LIN {X 0,Y 378.672,Z 1066.339,A -85,B 0,C 180,E1 1436.367,E2 1436.367} C_VEL
LIN {X 0,Y 367.013,Z 1084.806,A -85,B 0,C 180,E1 1435.562,E2 1435.562} C_VEL
LIN {X 0,Y 351.112,Z 1107.485,A -85,B 0,C 180,E1 1434.366,E2 1434.366} C_VEL
LIN {X 0,Y 334.229,Z 1128.583,A -85,B 0,C 180,E1 1432.955,E2 1432.955} C_VEL
LIN {X 0,Y 319.846,Z 1144.954,A -85,B 0,C 180,E1 1431.608,E2 1431.608} C_VEL
LIN {X 0,Y 305.454,Z 1160.008,A -85,B 0,C 180,E1 1430.12,E2 1430.12} C_VEL
LIN {X 0,Y 289.032,Z 1175.823,A -85,B 0,C 180,E1 1428.202,E2 1428.202} C_VEL
LIN {X 0,Y 267.713,Z 1194.413,A -85,B 0,C 180,E1 1425.283,E2 1425.283} C_VEL
LIN {X 0,Y 251.392,Z 1207.358,A -85,B 0,C 180,E1 1422.634,E2 1422.634} C_VEL
LIN {X 0,Y 235.673,Z 1218.959,A -85,B 0,C 180,E1 1419.631,E2 1419.631} C_VEL
LIN {X 0,Y 219.9,Z 1229.843,A -85,B 0,C 180,E1 1416.033,E2 1416.033} C_VEL
LIN {X 0,Y 201.548,Z 1241.771,A -85,B 0,C 180,E1 1410.804,E2 1410.804} C_VEL
LIN {X 0,Y 185.029,Z 1251.66,A -85,B 0,C 180,E1 1404.667,E2 1404.667} C_VEL
LIN {X 0,Y 172.413,Z 1259.033,A -85,B 0,C 180,E1 1398.41,E2 1398.41} C_VEL
LIN {X 0,Y 161.879,Z 1265.177,A -85,B 0,C 180,E1 1391.354,E2 1391.354} C_VEL
LIN {X 0,Y 152.21,Z 1271.176,A -85,B 0,C 180,E1 1381.69,E2 1381.69} C_VEL
LIN {X 0,Y 146.556,Z 1275.119,A -85,B 0,C 180,E1 1371.605,E2 1371.605} C_VEL
LIN {X 0,Y 144.431,Z 1277.221,A -85,B 0,C 180,E1 1363.194,E2 1363.194} C_VEL
LIN {X 0,Y 143.94,Z 1278.237,A -85,B 0,C 180,E1 1355.969,E2 1355.969} C_VEL
LIN {X 0,Y 143.895,Z 1278.557,A -85,B 0,C 180,E1 1349.59,E2 1349.59} C_VEL
LIN {X 0,Y 143.973,Z 1278.16,A -85,B 0,C 180,E1 1342.808,E2 1342.808} C_VEL
LIN {X 0,Y 145.059,Z 1276.539,A -85,B 0,C 180,E1 1333.362,E2 1333.362} C_VEL
LIN {X 0,Y 148.731,Z 1273.418,A -85,B 0,C 180,E1 1323.649,E2 1323.649} C_VEL
LIN {X 0,Y 154.712,Z 1269.457,A -85,B 0,C 180,E1 1315.327,E2 1315.327} C_VEL
LIN {X 0,Y 163.207,Z 1264.34,A -85,B 0,C 180,E1 1307.619,E2 1307.619} C_VEL
LIN {X 0,Y 174.045,Z 1258.034,A -85,B 0,C 180,E1 1300.67,E2 1300.67} C_VEL
LIN {X 0,Y 190.134,Z 1248.617,A -85,B 0,C 180,E1 1293.252,E2 1293.252} C_VEL
LIN {X 0,Y 206.536,Z 1238.422,A -85,B 0,C 180,E1 1287.62,E2 1287.62} C_VEL
LIN {X 0,Y 221.472,Z 1228.672,A -85,B 0,C 180,E1 1283.569,E2 1283.569} C_VEL
LIN {X 0,Y 237.335,Z 1217.651,A -85,B 0,C 180,E1 1280.02,E2 1280.02} C_VEL
LIN {X 0,Y 257.388,Z 1202.665,A -85,B 0,C 180,E1 1276.342,E2 1276.342} C_VEL
LIN {X 0,Y 276.552,Z 1186.732,A -85,B 0,C 180,E1 1273.434,E2 1273.434} C_VEL
LIN {X 0,Y 291.788,Z 1173.023,A -85,B 0,C 180,E1 1271.448,E2 1271.448} C_VEL
LIN {X 0,Y 307.342,Z 1157.869,A -85,B 0,C 180,E1 1269.664,E2 1269.664} C_VEL
LIN {X 0,Y 324.579,Z 1139.556,A -85,B 0,C 180,E1 1267.927,E2 1267.927} C_VEL
LIN {X 0,Y 342.558,Z 1118.091,A -85,B 0,C 180,E1 1266.322,E2 1266.322} C_VEL
LIN {X 0,Y 355.884,Z 1100.475,A -85,B 0,C 180,E1 1265.25,E2 1265.25} C_VEL
LIN {X 0,Y 368.516,Z 1082.112,A -85,B 0,C 180,E1 1264.318,E2 1264.318} C_VEL
LIN {X 0,Y 381.183,Z 1061.706,A -85,B 0,C 180,E1 1263.459,E2 1263.459} C_VEL
LIN {X 0,Y 395.364,Z 1035.586,A -85,B 0,C 180,E1 1262.573,E2 1262.573} C_VEL
LIN {X 0,Y 405.584,Z 1013.785,A -85,B 0,C 180,E1 1261.978,E2 1261.978} C_VEL
LIN {X 0,Y 413.929,Z 993.464,A -85,B 0,C 180,E1 1261.523,E2 1261.523} C_VEL
LIN {X 0,Y 421.543,Z 972.029,A -85,B 0,C 180,E1 1261.126,E2 1261.126} C_VEL
LIN {X 0,Y 429.495,Z 945.131,A -85,B 0,C 180,E1 1260.731,E2 1260.731} C_VEL
LIN {X 0,Y 435.377,Z 918.923,A -85,B 0,C 180,E1 1260.413,E2 1260.413} C_VEL
LIN {X 0,Y 439.185,Z 896.513,A -85,B 0,C 180,E1 1260.146,E2 1260.146} C_VEL
LIN {X 0,Y 441.739,Z 877.396,A -85,B 0,C 180,E1 1259.918,E2 1259.918} C_VEL
LIN {X 0,Y 436.632,Z 912.339,A -85,B 0,C 180,E1 1259.507,E2 1259.507} C_VEL
LIN {X 0,Y 431.778,Z 935.485,A -85,B 0,C 180,E1 1259.229,E2 1259.229} C_VEL
LIN {X 0,Y 426.116,Z 957.033,A -85,B 0,C 180,E1 1258.929,E2 1258.929} C_VEL
LIN {X 0,Y 418.849,Z 979.936,A -85,B 0,C 180,E1 1258.534,E2 1258.534} C_VEL
LIN {X 0,Y 408.228,Z 1007.518,A -85,B 0,C 180,E1 1257.937,E2 1257.937} C_VEL
LIN {X 0,Y 398.391,Z 1029.133,A -85,B 0,C 180,E1 1257.352,E2 1257.352} C_VEL
LIN {X 0,Y 388.597,Z 1048.173,A -85,B 0,C 180,E1 1256.736,E2 1256.736} C_VEL
LIN {X 0,Y 377.878,Z 1066.847,A -85,B 0,C 180,E1 1256.025,E2 1256.025} C_VEL
LIN {X 0,Y 365.295,Z 1086.576,A -85,B 0,C 180,E1 1255.12,E2 1255.12} C_VEL
LIN {X 0,Y 348.427,Z 1110.03,A -85,B 0,C 180,E1 1253.806,E2 1253.806} C_VEL
LIN {X 0,Y 333.793,Z 1128.151,A -85,B 0,C 180,E1 1252.551,E2 1252.551} C_VEL
LIN {X 0,Y 319.333,Z 1144.499,A -85,B 0,C 180,E1 1251.174,E2 1251.174} C_VEL
LIN {X 0,Y 304.427,Z 1159.961,A -85,B 0,C 180,E1 1249.592,E2 1249.592} C_VEL
LIN {X 0,Y 285.915,Z 1177.579,A -85,B 0,C 180,E1 1247.359,E2 1247.359} C_VEL
LIN {X 0,Y 266.517,Z 1194.056,A -85,B 0,C 180,E1 1244.632,E2 1244.632} C_VEL
LIN {X 0,Y 250.312,Z 1206.744,A -85,B 0,C 180,E1 1241.948,E2 1241.948} C_VEL
LIN {X 0,Y 234.708,Z 1218.094,A -85,B 0,C 180,E1 1238.915,E2 1238.915} C_VEL
LIN {X 0,Y 216.804,Z 1230.255,A -85,B 0,C 180,E1 1234.693,E2 1234.693} C_VEL
LIN {X 0,Y 198.115,Z 1241.878,A -85,B 0,C 180,E1 1229.103,E2 1229.103} C_VEL
LIN {X 0,Y 184.307,Z 1250.012,A -85,B 0,C 180,E1 1223.748,E2 1223.748} C_VEL
LIN {X 0,Y 172.154,Z 1256.949,A -85,B 0,C 180,E1 1217.643,E2 1217.643} C_VEL
LIN {X 0,Y 161.235,Z 1263.175,A -85,B 0,C 180,E1 1210.173,E2 1210.173} C_VEL
LIN {X 0,Y 151.586,Z 1268.911,A -85,B 0,C 180,E1 1200.098,E2 1200.098} C_VEL
LIN {X 0,Y 146.712,Z 1272.204,A -85,B 0,C 180,E1 1191.186,E2 1191.186} C_VEL
LIN {X 0,Y 144.596,Z 1274.118,A -85,B 0,C 180,E1 1183.202,E2 1183.202} C_VEL
LIN {X 0,Y 143.969,Z 1275.117,A -85,B 0,C 180,E1 1175.591,E2 1175.591} C_VEL
LIN {X 0,Y 143.896,Z 1275.371,A -85,B 0,C 180,E1 1168.817,E2 1168.817} C_VEL
LIN {X 0,Y 144.083,Z 1274.947,A -85,B 0,C 180,E1 1161.632,E2 1161.632} C_VEL
LIN {X 0,Y 145.518,Z 1273.259,A -85,B 0,C 180,E1 1152.415,E2 1152.415} C_VEL
LIN {X 0,Y 149.301,Z 1270.396,A -85,B 0,C 180,E1 1143.353,E2 1143.353} C_VEL
LIN {X 0,Y 155.5,Z 1266.534,A -85,B 0,C 180,E1 1135.105,E2 1135.105} C_VEL
LIN {X 0,Y 163.722,Z 1261.781,A -85,B 0,C 180,E1 1127.81,E2 1127.81} C_VEL
LIN {X 0,Y 174.598,Z 1255.648,A -85,B 0,C 180,E1 1120.91,E2 1120.91} C_VEL
LIN {X 0,Y 190.038,Z 1246.867,A -85,B 0,C 180,E1 1113.785,E2 1113.785} C_VEL
LIN {X 0,Y 207.134,Z 1236.43,A -85,B 0,C 180,E1 1107.921,E2 1107.921} C_VEL
LIN {X 0,Y 221.976,Z 1226.888,A -85,B 0,C 180,E1 1103.902,E2 1103.902} C_VEL
LIN {X 0,Y 237.791,Z 1216.047,A -85,B 0,C 180,E1 1100.36,E2 1100.36} C_VEL
LIN {X 0,Y 256.926,Z 1201.952,A -85,B 0,C 180,E1 1096.822,E2 1096.822} C_VEL
LIN {X 0,Y 276.577,Z 1185.833,A -85,B 0,C 180,E1 1093.804,E2 1093.804} C_VEL
LIN {X 0,Y 292.07,Z 1172.028,A -85,B 0,C 180,E1 1091.773,E2 1091.773} C_VEL
LIN {X 0,Y 307.577,Z 1157.038,A -85,B 0,C 180,E1 1089.98,E2 1089.98} C_VEL
LIN {X 0,Y 323.353,Z 1140.42,A -85,B 0,C 180,E1 1088.356,E2 1088.356} C_VEL
LIN {X 0,Y 342.209,Z 1118.276,A -85,B 0,C 180,E1 1086.635,E2 1086.635} C_VEL
LIN {X 0,Y 356.327,Z 1099.724,A -85,B 0,C 180,E1 1085.475,E2 1085.475} C_VEL
LIN {X 0,Y 369.062,Z 1081.271,A -85,B 0,C 180,E1 1084.523,E2 1084.523} C_VEL
LIN {X 0,Y 381.194,Z 1061.783,A -85,B 0,C 180,E1 1083.673,E2 1083.673} C_VEL
LIN {X 0,Y 395.463,Z 1035.672,A -85,B 0,C 180,E1 1082.754,E2 1082.754} C_VEL
LIN {X 0,Y 405.737,Z 1013.852,A -85,B 0,C 180,E1 1082.131,E2 1082.131} C_VEL
LIN {X 0,Y 414.382,Z 992.844,A -85,B 0,C 180,E1 1081.635,E2 1081.635} C_VEL
LIN {X 0,Y 422.249,Z 970.633,A -85,B 0,C 180,E1 1081.202,E2 1081.202} C_VEL
LIN {X 0,Y 430.583,Z 941.674,A -85,B 0,C 180,E1 1080.76,E2 1080.76} C_VEL
LIN {X 0,Y 435.823,Z 918.039,A -85,B 0,C 180,E1 1080.47,E2 1080.47} C_VEL
LIN {X 0,Y 439.576,Z 895.786,A -85,B 0,C 180,E1 1080.207,E2 1080.207} C_VEL
LIN {X 0,Y 441.526,Z 881.472,A -85,B 0,C 180,E1 1080.03,E2 1080.03} C_VEL
LIN {X 0,Y 438.256,Z 904.869,A -85,B 0,C 180,E1 1079.756,E2 1079.756} C_VEL
LIN {X 0,Y 438.232,Z 905.207,A -85,B 0,C 180,E1 1079.754,E2 1079.754} C_VEL
LIN {X 0,Y 438.232,Z 987.285,A -85,B 0,C 180,E1 1079.754,E2 1079.754} C_VEL
LIN {X 0,Y 429.018,Z 987.285,A -85,B 0,C 180,E1 1080.138,E2 1080.138} C_VEL
LIN {X 0,Y 427.112,Z 985.285,A -85,B 0,C 180,E1 1080.219,E2 1080.219} C_VEL
LIN {X 0,Y 427.112,Z 967.597,A -85,B 0,C 180,E1 1080.219,E2 1080.219} C_VEL
LIN {X 0,Y 423.438,Z 966.924,A -85,B 0,C 180,E1 1080.05,E2 1080.05} C_VEL
LIN {X 0,Y 414.913,Z 991.21,A -85,B 0,C 180,E1 1079.638,E2 1079.638} C_VEL
LIN {X 0,Y 406.365,Z 1012.095,A -85,B 0,C 180,E1 1079.204,E2 1079.204} C_VEL
LIN {X 0,Y 397.01,Z 1032.135,A -85,B 0,C 180,E1 1078.701,E2 1078.701} C_VEL
LIN {X 0,Y 385.683,Z 1053.594,A -85,B 0,C 180,E1 1078.049,E2 1078.049} C_VEL
LIN {X 0,Y 370.387,Z 1078.828,A -85,B 0,C 180,E1 1077.098,E2 1077.098} C_VEL
LIN {X 0,Y 356.715,Z 1098.707,A -85,B 0,C 180,E1 1076.161,E2 1076.161} C_VEL
LIN {X 0,Y 343.626,Z 1115.951,A -85,B 0,C 180,E1 1075.191,E2 1075.191} C_VEL
LIN {X 0,Y 328.734,Z 1133.826,A -85,B 0,C 180,E1 1073.976,E2 1073.976} C_VEL
LIN {X 0,Y 308.826,Z 1155.272,A -85,B 0,C 180,E1 1072.137,E2 1072.137} C_VEL
LIN {X 0,Y 291.848,Z 1171.676,A -85,B 0,C 180,E1 1070.336,E2 1070.336} C_VEL
LIN {X 0,Y 276.499,Z 1185.321,A -85,B 0,C 180,E1 1068.479,E2 1068.479} C_VEL
LIN {X 0,Y 260.39,Z 1198.549,A -85,B 0,C 180,E1 1066.253,E2 1066.253} C_VEL
LIN {X 0,Y 240.461,Z 1213.656,A -85,B 0,C 180,E1 1062.984,E2 1062.984} C_VEL
LIN {X 0,Y 220.609,Z 1227.16,A -85,B 0,C 180,E1 1058.987,E2 1058.987} C_VEL
LIN {X 0,Y 204.239,Z 1237.526,A -85,B 0,C 180,E1 1054.893,E2 1054.893} C_VEL
LIN {X 0,Y 189.028,Z 1246.591,A -85,B 0,C 180,E1 1050.147,E2 1050.147} C_VEL
LIN {X 0,Y 172.191,Z 1256.182,A -85,B 0,C 180,E1 1043.239,E2 1043.239} C_VEL
LIN {X 0,Y 158.056,Z 1263.798,A -85,B 0,C 180,E1 1035.098,E2 1035.098} C_VEL
LIN {X 0,Y 148.642,Z 1268.998,A -85,B 0,C 180,E1 1027.243,E2 1027.243} C_VEL
LIN {X 0,Y 142.104,Z 1272.88,A -85,B 0,C 180,E1 1019.031,E2 1019.031} C_VEL
LIN {X 0,Y 138.152,Z 1275.61,A -85,B 0,C 180,E1 1010.758,E2 1010.758} C_VEL
LIN {X 0,Y 136.348,Z 1277.342,A -85,B 0,C 180,E1 1002.696,E2 1002.696} C_VEL
LIN {X 0,Y 135.93,Z 1278.196,A -85,B 0,C 180,E1 995.475,E2 995.475} C_VEL
LIN {X 0,Y 135.897,Z 1278.424,A -85,B 0,C 180,E1 988.723,E2 988.723} C_VEL
LIN {X 0,Y 136,Z 1278.016,A -85,B 0,C 180,E1 981.533,E2 981.533} C_VEL
LIN {X 0,Y 137.407,Z 1276.277,A -85,B 0,C 180,E1 971.754,E2 971.754} C_VEL
LIN {X 0,Y 141.403,Z 1273.309,A -85,B 0,C 180,E1 962.117,E2 962.117} C_VEL
LIN {X 0,Y 147.936,Z 1269.365,A -85,B 0,C 180,E1 953.491,E2 953.491} C_VEL
LIN {X 0,Y 157.124,Z 1264.248,A -85,B 0,C 180,E1 945.56,E2 945.56} C_VEL
LIN {X 0,Y 168.742,Z 1257.911,A -85,B 0,C 180,E1 938.476,E2 938.476} C_VEL
LIN {X 0,Y 185.648,Z 1248.524,A -85,B 0,C 180,E1 931.077,E2 931.077} C_VEL
LIN {X 0,Y 202.77,Z 1238.328,A -85,B 0,C 180,E1 925.511,E2 925.511} C_VEL
LIN {X 0,Y 218.581,Z 1228.359,A -85,B 0,C 180,E1 921.467,E2 921.467} C_VEL
LIN {X 0,Y 234.592,Z 1217.557,A -85,B 0,C 180,E1 918.092,E2 918.092} C_VEL
LIN {X 0,Y 255.158,Z 1202.572,A -85,B 0,C 180,E1 914.537,E2 914.537} C_VEL
LIN {X 0,Y 274.734,Z 1186.638,A -85,B 0,C 180,E1 911.74,E2 911.74} C_VEL
LIN {X 0,Y 290.25,Z 1172.929,A -85,B 0,C 180,E1 909.836,E2 909.836} C_VEL
LIN {X 0,Y 306.056,Z 1157.775,A -85,B 0,C 180,E1 908.13,E2 908.13} C_VEL
LIN {X 0,Y 323.416,Z 1139.596,A -85,B 0,C 180,E1 906.485,E2 906.485} C_VEL
LIN {X 0,Y 341.515,Z 1118.293,A -85,B 0,C 180,E1 904.967,E2 904.967} C_VEL
LIN {X 0,Y 355.307,Z 1100.272,A -85,B 0,C 180,E1 903.928,E2 903.928} C_VEL
LIN {X 0,Y 367.913,Z 1082.134,A -85,B 0,C 180,E1 903.053,E2 903.053} C_VEL
LIN {X 0,Y 380.265,Z 1062.458,A -85,B 0,C 180,E1 902.265,E2 902.265} C_VEL
LIN {X 0,Y 394.588,Z 1036.497,A -85,B 0,C 180,E1 901.425,E2 901.425} C_VEL
LIN {X 0,Y 405.119,Z 1014.297,A -85,B 0,C 180,E1 900.849,E2 900.849} C_VEL
LIN {X 0,Y 413.579,Z 993.918,A -85,B 0,C 180,E1 900.416,E2 900.416} C_VEL
LIN {X 0,Y 420.962,Z 973.413,A -85,B 0,C 180,E1 900.054,E2 900.054} C_VEL
LIN {X 0,Y 424.03,Z 964.106,A -85,B 0,C 180,E1 899.903,E2 899.903} C_VEL
LIN {X 0,Y 414.982,Z 990.252,A -85,B 0,C 180,E1 899.442,E2 899.442} C_VEL
LIN {X 0,Y 406.528,Z 1010.997,A -85,B 0,C 180,E1 898.989,E2 898.989} C_VEL
LIN {X 0,Y 397.109,Z 1031.233,A -85,B 0,C 180,E1 898.458,E2 898.458} C_VEL
LIN {X 0,Y 386.249,Z 1051.858,A -85,B 0,C 180,E1 897.811,E2 897.811} C_VEL
LIN {X 0,Y 371.525,Z 1076.416,A -85,B 0,C 180,E1 896.867,E2 896.867} C_VEL
LIN {X 0,Y 357.524,Z 1096.849,A -85,B 0,C 180,E1 895.894,E2 895.894} C_VEL
LIN {X 0,Y 344.342,Z 1114.269,A -85,B 0,C 180,E1 894.892,E2 894.892} C_VEL
LIN {X 0,Y 330.395,Z 1131.062,A -85,B 0,C 180,E1 893.745,E2 893.745} C_VEL
LIN {X 0,Y 313.589,Z 1149.501,A -85,B 0,C 180,E1 892.202,E2 892.202} C_VEL
LIN {X 0,Y 294.291,Z 1168.425,A -85,B 0,C 180,E1 890.184,E2 890.184} C_VEL
LIN {X 0,Y 277.332,Z 1183.499,A -85,B 0,C 180,E1 888.141,E2 888.141} C_VEL
LIN {X 0,Y 261.779,Z 1196.239,A -85,B 0,C 180,E1 885.987,E2 885.987} C_VEL
LIN {X 0,Y 245.282,Z 1208.73,A -85,B 0,C 180,E1 883.345,E2 883.345} C_VEL
LIN {X 0,Y 225.194,Z 1222.744,A -85,B 0,C 180,E1 879.465,E2 879.465} C_VEL
LIN {X 0,Y 206.425,Z 1234.551,A -85,B 0,C 180,E1 874.944,E2 874.944} C_VEL
LIN {X 0,Y 191.824,Z 1243.174,A -85,B 0,C 180,E1 870.528,E2 870.528} C_VEL
LIN {X 0,Y 177.813,Z 1251.022,A -85,B 0,C 180,E1 865.197,E2 865.197} C_VEL
LIN {X 0,Y 163.802,Z 1258.601,A -85,B 0,C 180,E1 858.147,E2 858.147} C_VEL
LIN {X 0,Y 150.561,Z 1265.616,A -85,B 0,C 180,E1 848.404,E2 848.404} C_VEL
LIN {X 0,Y 143.078,Z 1269.786,A -85,B 0,C 180,E1 839.759,E2 839.759} C_VEL
LIN {X 0,Y 138.77,Z 1272.517,A -85,B 0,C 180,E1 831.572,E2 831.572} C_VEL
LIN {X 0,Y 136.638,Z 1274.273,A -85,B 0,C 180,E1 823.554,E2 823.554} C_VEL
LIN {X 0,Y 135.98,Z 1275.205,A -85,B 0,C 180,E1 815.921,E2 815.921} C_VEL
LIN {X 0,Y 135.894,Z 1275.481,A -85,B 0,C 180,E1 809.169,E2 809.169} C_VEL
LIN {X 0,Y 136.071,Z 1275.108,A -85,B 0,C 180,E1 801.987,E2 801.987} C_VEL
LIN {X 0,Y 137.524,Z 1273.57,A -85,B 0,C 180,E1 792.233,E2 792.233} C_VEL
LIN {X 0,Y 141.736,Z 1270.643,A -85,B 0,C 180,E1 782.265,E2 782.265} C_VEL
LIN {X 0,Y 148.399,Z 1266.828,A -85,B 0,C 180,E1 773.651,E2 773.651} C_VEL
LIN {X 0,Y 157.642,Z 1261.872,A -85,B 0,C 180,E1 765.774,E2 765.774} C_VEL
LIN {X 0,Y 169.236,Z 1255.738,A -85,B 0,C 180,E1 758.769,E2 758.769} C_VEL
LIN {X 0,Y 186.188,Z 1246.556,A -85,B 0,C 180,E1 751.385,E2 751.385} C_VEL
LIN {X 0,Y 203.277,Z 1236.557,A -85,B 0,C 180,E1 745.847,E2 745.847} C_VEL
LIN {X 0,Y 218.711,Z 1226.979,A -85,B 0,C 180,E1 741.892,E2 741.892} C_VEL
LIN {X 0,Y 235.009,Z 1216.137,A -85,B 0,C 180,E1 738.446,E2 738.446} C_VEL
LIN {X 0,Y 254.654,Z 1202.027,A -85,B 0,C 180,E1 735.02,E2 735.02} C_VEL
LIN {X 0,Y 274.117,Z 1186.428,A -85,B 0,C 180,E1 732.197,E2 732.197} C_VEL
LIN {X 0,Y 290.489,Z 1172.116,A -85,B 0,C 180,E1 730.169,E2 730.169} C_VEL
LIN {X 0,Y 306.322,Z 1157.055,A -85,B 0,C 180,E1 728.447,E2 728.447} C_VEL
LIN {X 0,Y 322.821,Z 1139.909,A -85,B 0,C 180,E1 726.856,E2 726.856} C_VEL
LIN {X 0,Y 341.358,Z 1118.362,A -85,B 0,C 180,E1 725.267,E2 725.267} C_VEL
LIN {X 0,Y 355.164,Z 1100.462,A -85,B 0,C 180,E1 724.198,E2 724.198} C_VEL
LIN {X 0,Y 368.02,Z 1082.087,A -85,B 0,C 180,E1 723.292,E2 723.292} C_VEL
LIN {X 0,Y 379.791,Z 1063.462,A -85,B 0,C 180,E1 722.513,E2 722.513} C_VEL
LIN {X 0,Y 393.082,Z 1039.924,A -85,B 0,C 180,E1 721.704,E2 721.704} C_VEL
LIN {X 0,Y 404.971,Z 1015.175,A -85,B 0,C 180,E1 721.021,E2 721.021} C_VEL
LIN {X 0,Y 413.592,Z 994.567,A -85,B 0,C 180,E1 720.554,E2 720.554} C_VEL
LIN {X 0,Y 420.906,Z 974.413,A -85,B 0,C 180,E1 720.173,E2 720.173} C_VEL
LIN {X 0,Y 423.438,Z 966.924,A -85,B 0,C 180,E1 720.05,E2 720.05} C_VEL
LIN {X 0,Y 427.11,Z 967.598,A -85,B 0,C 180,E1 719.88,E2 719.88} C_VEL
LIN {X 0,Y 427.11,Z 1038.968,A -85,B 0,C 180,E1 719.88,E2 719.88} C_VEL
LIN {X 0,Y 406.612,Z 1038.968,A -85,B 0,C 180,E1 720.222,E2 720.222} C_VEL
LIN {X 0,Y 404.627,Z 1036.968,A -85,B 0,C 180,E1 720.257,E2 720.257} C_VEL
LIN {X 0,Y 404.627,Z 1024.614,A -85,B 0,C 180,E1 720.257,E2 720.257} C_VEL
LIN {X 0,Y 401.065,Z 1023.683,A -85,B 0,C 180,E1 720.081,E2 720.081} C_VEL
LIN {X 0,Y 389.299,Z 1046.613,A -85,B 0,C 180,E1 719.468,E2 719.468} C_VEL
LIN {X 0,Y 378.485,Z 1065.358,A -85,B 0,C 180,E1 718.863,E2 718.863} C_VEL
LIN {X 0,Y 366.555,Z 1083.973,A -85,B 0,C 180,E1 718.146,E2 718.146} C_VEL
LIN {X 0,Y 352.332,Z 1103.977,A -85,B 0,C 180,E1 717.214,E2 717.214} C_VEL
LIN {X 0,Y 333.788,Z 1127.058,A -85,B 0,C 180,E1 715.863,E2 715.863} C_VEL
LIN {X 0,Y 318.812,Z 1143.762,A -85,B 0,C 180,E1 714.645,E2 714.645} C_VEL
LIN {X 0,Y 303.519,Z 1159.367,A -85,B 0,C 180,E1 713.263,E2 713.263} C_VEL
LIN {X 0,Y 287.024,Z 1174.797,A -85,B 0,C 180,E1 711.574,E2 711.574} C_VEL
LIN {X 0,Y 266.693,Z 1192.121,A -85,B 0,C 180,E1 709.155,E2 709.155} C_VEL
LIN {X 0,Y 246.904,Z 1207.179,A -85,B 0,C 180,E1 706.353,E2 706.353} C_VEL
LIN {X 0,Y 230.362,Z 1218.779,A -85,B 0,C 180,E1 703.553,E2 703.553} C_VEL
LIN {X 0,Y 213.616,Z 1229.662,A -85,B 0,C 180,E1 700.162,E2 700.162} C_VEL
LIN {X 0,Y 193.881,Z 1241.589,A -85,B 0,C 180,E1 695.16,E2 695.16} C_VEL
LIN {X 0,Y 175.841,Z 1251.478,A -85,B 0,C 180,E1 689.141,E2 689.141} C_VEL
LIN {X 0,Y 161.747,Z 1258.851,A -85,B 0,C 180,E1 682.867,E2 682.867} C_VEL
LIN {X 0,Y 149.729,Z 1264.995,A -85,B 0,C 180,E1 675.587,E2 675.587} C_VEL
LIN {X 0,Y 138.298,Z 1271.033,A -85,B 0,C 180,E1 665.216,E2 665.216} C_VEL
LIN {X 0,Y 131.277,Z 1275.021,A -85,B 0,C 180,E1 653.936,E2 653.936} C_VEL
LIN {X 0,Y 128.652,Z 1277.043,A -85,B 0,C 180,E1 644.847,E2 644.847} C_VEL
LIN {X 0,Y 127.959,Z 1278.061,A -85,B 0,C 180,E1 636.718,E2 636.718} C_VEL
LIN {X 0,Y 127.895,Z 1278.382,A -85,B 0,C 180,E1 629.539,E2 629.539} C_VEL
LIN {X 0,Y 127.986,Z 1278.007,A -85,B 0,C 180,E1 622.355,E2 622.355} C_VEL
LIN {X 0,Y 129.309,Z 1276.528,A -85,B 0,C 180,E1 611.97,E2 611.97} C_VEL
LIN {X 0,Y 134.125,Z 1273.236,A -85,B 0,C 180,E1 600.514,E2 600.514} C_VEL
LIN {X 0,Y 141.321,Z 1269.273,A -85,B 0,C 180,E1 591.479,E2 591.479} C_VEL
LIN {X 0,Y 150.964,Z 1264.303,A -85,B 0,C 180,E1 583.538,E2 583.538} C_VEL
LIN {X 0,Y 162.979,Z 1258.155,A -85,B 0,C 180,E1 576.502,E2 576.502} C_VEL
LIN {X 0,Y 180.266,Z 1249.109,A -85,B 0,C 180,E1 569.217,E2 569.217} C_VEL
LIN {X 0,Y 199.291,Z 1238.235,A -85,B 0,C 180,E1 563.328,E2 563.328} C_VEL
LIN {X 0,Y 215.298,Z 1228.484,A -85,B 0,C 180,E1 559.462,E2 559.462} C_VEL
LIN {X 0,Y 232.121,Z 1217.463,A -85,B 0,C 180,E1 556.121,E2 556.121} C_VEL
LIN {X 0,Y 252.408,Z 1203.074,A -85,B 0,C 180,E1 552.817,E2 552.817} C_VEL
LIN {X 0,Y 272.238,Z 1187.318,A -85,B 0,C 180,E1 550.139,E2 550.139} C_VEL
LIN {X 0,Y 288.007,Z 1173.684,A -85,B 0,C 180,E1 548.31,E2 548.31} C_VEL
LIN {X 0,Y 304.043,Z 1158.611,A -85,B 0,C 180,E1 546.677,E2 546.677} C_VEL
LIN {X 0,Y 319.824,Z 1142.421,A -85,B 0,C 180,E1 545.258,E2 545.258} C_VEL
LIN {X 0,Y 338.216,Z 1121.566,A -85,B 0,C 180,E1 543.793,E2 543.793} C_VEL
LIN {X 0,Y 353.667,Z 1101.777,A -85,B 0,C 180,E1 542.685,E2 542.685} C_VEL
LIN {X 0,Y 366.659,Z 1083.397,A -85,B 0,C 180,E1 541.836,E2 541.836} C_VEL
LIN {X 0,Y 378.541,Z 1064.803,A -85,B 0,C 180,E1 541.122,E2 541.122} C_VEL
LIN {X 0,Y 390.529,Z 1043.878,A -85,B 0,C 180,E1 540.455,E2 540.455} C_VEL
LIN {X 0,Y 401.702,Z 1021.82,A -85,B 0,C 180,E1 539.873,E2 539.873} C_VEL
LIN {X 0,Y 389.503,Z 1045.669,A -85,B 0,C 180,E1 539.213,E2 539.213} C_VEL
LIN {X 0,Y 378.585,Z 1064.608,A -85,B 0,C 180,E1 538.581,E2 538.581} C_VEL
LIN {X 0,Y 366.681,Z 1083.175,A -85,B 0,C 180,E1 537.838,E2 537.838} C_VEL
LIN {X 0,Y 353.47,Z 1101.782,A -85,B 0,C 180,E1 536.959,E2 536.959} C_VEL
LIN {X 0,Y 335.936,Z 1123.914,A -85,B 0,C 180,E1 535.665,E2 535.665} C_VEL
LIN {X 0,Y 319.021,Z 1142.792,A -85,B 0,C 180,E1 534.272,E2 534.272} C_VEL
LIN {X 0,Y 304.3,Z 1157.787,A -85,B 0,C 180,E1 532.921,E2 532.921} C_VEL
LIN {X 0,Y 289.249,Z 1171.882,A -85,B 0,C 180,E1 531.382,E2 531.382} C_VEL
LIN {X 0,Y 272.43,Z 1186.359,A -85,B 0,C 180,E1 529.425,E2 529.425} C_VEL
LIN {X 0,Y 251.834,Z 1202.514,A -85,B 0,C 180,E1 526.611,E2 526.611} C_VEL
LIN {X 0,Y 232.626,Z 1216.004,A -85,B 0,C 180,E1 523.454,E2 523.454} C_VEL
LIN {X 0,Y 215.86,Z 1226.867,A -85,B 0,C 180,E1 520.12,E2 520.12} C_VEL
LIN {X 0,Y 199.897,Z 1236.463,A -85,B 0,C 180,E1 516.272,E2 516.272} C_VEL
LIN {X 0,Y 181.393,Z 1246.876,A -85,B 0,C 180,E1 510.582,E2 510.582} C_VEL
LIN {X 0,Y 163.758,Z 1255.939,A -85,B 0,C 180,E1 503.246,E2 503.246} C_VEL
LIN {X 0,Y 151.441,Z 1262.072,A -85,B 0,C 180,E1 496.111,E2 496.111} C_VEL
LIN {X 0,Y 141.49,Z 1267.031,A -85,B 0,C 180,E1 487.951,E2 487.951} C_VEL
LIN {X 0,Y 133.06,Z 1271.598,A -85,B 0,C 180,E1 476.812,E2 476.812} C_VEL
LIN {X 0,Y 129.025,Z 1274.164,A -85,B 0,C 180,E1 465.75,E2 465.75} C_VEL
LIN {X 0,Y 128.012,Z 1275.272,A -85,B 0,C 180,E1 456.741,E2 456.741} C_VEL
LIN {X 0,Y 127.898,Z 1275.591,A -85,B 0,C 180,E1 449.565,E2 449.565} C_VEL
LIN {X 0,Y 128.072,Z 1275.217,A -85,B 0,C 180,E1 441.935,E2 441.935} C_VEL
LIN {X 0,Y 129.663,Z 1273.759,A -85,B 0,C 180,E1 431.534,E2 431.534} C_VEL
LIN {X 0,Y 134.493,Z 1270.733,A -85,B 0,C 180,E1 420.63,E2 420.63} C_VEL
LIN {X 0,Y 142.093,Z 1266.762,A -85,B 0,C 180,E1 411.361,E2 411.361} C_VEL
LIN {X 0,Y 151.774,Z 1261.962,A -85,B 0,C 180,E1 403.576,E2 403.576} C_VEL
LIN {X 0,Y 164.121,Z 1255.829,A -85,B 0,C 180,E1 396.488,E2 396.488} C_VEL
LIN {X 0,Y 181.259,Z 1247.047,A -85,B 0,C 180,E1 389.38,E2 389.38} C_VEL
LIN {X 0,Y 199.762,Z 1236.647,A -85,B 0,C 180,E1 383.68,E2 383.68} C_VEL
LIN {X 0,Y 216.128,Z 1226.818,A -85,B 0,C 180,E1 379.738,E2 379.738} C_VEL
LIN {X 0,Y 233.353,Z 1215.657,A -85,B 0,C 180,E1 376.334,E2 376.334} C_VEL
LIN {X 0,Y 254.384,Z 1200.784,A -85,B 0,C 180,E1 372.932,E2 372.932} C_VEL
LIN {X 0,Y 273.398,Z 1185.75,A -85,B 0,C 180,E1 370.374,E2 370.374} C_VEL
LIN {X 0,Y 289.139,Z 1172.204,A -85,B 0,C 180,E1 368.55,E2 368.55} C_VEL
LIN {X 0,Y 305.144,Z 1157.213,A -85,B 0,C 180,E1 366.917,E2 366.917} C_VEL
LIN {X 0,Y 321.372,Z 1140.593,A -85,B 0,C 180,E1 365.448,E2 365.448} C_VEL
LIN {X 0,Y 340.703,Z 1118.448,A -85,B 0,C 180,E1 363.893,E2 363.893} C_VEL
LIN {X 0,Y 354.859,Z 1100.276,A -85,B 0,C 180,E1 362.866,E2 362.866} C_VEL
LIN {X 0,Y 367.565,Z 1082.287,A -85,B 0,C 180,E1 362.027,E2 362.027} C_VEL
LIN {X 0,Y 379.506,Z 1063.57,A -85,B 0,C 180,E1 361.287,E2 361.287} C_VEL
LIN {X 0,Y 392.925,Z 1040.007,A -85,B 0,C 180,E1 360.523,E2 360.523} C_VEL
LIN {X 0,Y 401.065,Z 1023.683,A -85,B 0,C 180,E1 360.081,E2 360.081} C_VEL
LIN {X 0,Y 404.622,Z 1024.617,A -85,B 0,C 180,E1 359.904,E2 359.904} C_VEL
LIN {X 0,Y 404.622,Z 1078.491,A -85,B 0,C 180,E1 359.904,E2 359.904} C_VEL
LIN {X 0,Y 383.996,Z 1078.491,A -85,B 0,C 180,E1 360.259,E2 360.259} C_VEL
LIN {X 0,Y 382.01,Z 1076.491,A -85,B 0,C 180,E1 360.295,E2 360.295} C_VEL
LIN {X 0,Y 382.01,Z 1066.132,A -85,B 0,C 180,E1 360.295,E2 360.295} C_VEL
LIN {X 0,Y 378.557,Z 1065.037,A -85,B 0,C 180,E1 360.106,E2 360.106} C_VEL
LIN {X 0,Y 366.621,Z 1083.533,A -85,B 0,C 180,E1 359.439,E2 359.439} C_VEL
LIN {X 0,Y 353.019,Z 1102.552,A -85,B 0,C 180,E1 358.609,E2 358.609} C_VEL
LIN {X 0,Y 334.768,Z 1125.301,A -85,B 0,C 180,E1 357.38,E2 357.38} C_VEL
LIN {X 0,Y 318.632,Z 1143.167,A -85,B 0,C 180,E1 356.169,E2 356.169} C_VEL
LIN {X 0,Y 303.138,Z 1158.815,A -85,B 0,C 180,E1 354.868,E2 354.868} C_VEL
LIN {X 0,Y 286.873,Z 1173.859,A -85,B 0,C 180,E1 353.32,E2 353.32} C_VEL
LIN {X 0,Y 267.111,Z 1190.563,A -85,B 0,C 180,E1 351.148,E2 351.148} C_VEL
LIN {X 0,Y 245.968,Z 1206.45,A -85,B 0,C 180,E1 348.387,E2 348.387} C_VEL
LIN {X 0,Y 229.006,Z 1218.112,A -85,B 0,C 180,E1 345.726,E2 345.726} C_VEL
LIN {X 0,Y 212.601,Z 1228.535,A -85,B 0,C 180,E1 342.66,E2 342.66} C_VEL
LIN {X 0,Y 195.267,Z 1238.732,A -85,B 0,C 180,E1 338.711,E2 338.711} C_VEL
LIN {X 0,Y 175.294,Z 1249.603,A -85,B 0,C 180,E1 332.826,E2 332.826} C_VEL
LIN {X 0,Y 158.093,Z 1258.147,A -85,B 0,C 180,E1 325.926,E2 325.926} C_VEL
LIN {X 0,Y 145.058,Z 1264.389,A -85,B 0,C 180,E1 318.686,E2 318.686} C_VEL
LIN {X 0,Y 134.45,Z 1269.446,A -85,B 0,C 180,E1 310.298,E2 310.298} C_VEL
LIN {X 0,Y 125.855,Z 1273.838,A -85,B 0,C 180,E1 299.493,E2 299.493} C_VEL
LIN {X 0,Y 121.09,Z 1276.744,A -85,B 0,C 180,E1 287.278,E2 287.278} C_VEL
LIN {X 0,Y 119.971,Z 1277.973,A -85,B 0,C 180,E1 277.168,E2 277.168} C_VEL
LIN {X 0,Y 119.896,Z 1278.294,A -85,B 0,C 180,E1 269.508,E2 269.508} C_VEL
LIN {X 0,Y 119.991,Z 1277.919,A -85,B 0,C 180,E1 261.843,E2 261.843} C_VEL
LIN {X 0,Y 121.437,Z 1276.513,A -85,B 0,C 180,E1 251.243,E2 251.243} C_VEL
LIN {X 0,Y 126.703,Z 1273.308,A -85,B 0,C 180,E1 239.126,E2 239.126} C_VEL
LIN {X 0,Y 134.473,Z 1269.391,A -85,B 0,C 180,E1 229.678,E2 229.678} C_VEL
LIN {X 0,Y 145.086,Z 1264.321,A -85,B 0,C 180,E1 221.292,E2 221.292} C_VEL
LIN {X 0,Y 157.485,Z 1258.368,A -85,B 0,C 180,E1 214.358,E2 214.358} C_VEL
LIN {X 0,Y 173.317,Z 1250.492,A -85,B 0,C 180,E1 207.859,E2 207.859} C_VEL
LIN {X 0,Y 194.505,Z 1239.066,A -85,B 0,C 180,E1 201.476,E2 201.476} C_VEL
LIN {X 0,Y 211.797,Z 1228.909,A -85,B 0,C 180,E1 197.498,E2 197.498} C_VEL
LIN {X 0,Y 228.171,Z 1218.524,A -85,B 0,C 180,E1 194.409,E2 194.409} C_VEL
LIN {X 0,Y 246.014,Z 1206.26,A -85,B 0,C 180,E1 191.599,E2 191.599} C_VEL
LIN {X 0,Y 268.091,Z 1189.548,A -85,B 0,C 180,E1 188.727,E2 188.727} C_VEL
LIN {X 0,Y 286.923,Z 1173.591,A -85,B 0,C 180,E1 186.666,E2 186.666} C_VEL
LIN {X 0,Y 303.19,Z 1158.517,A -85,B 0,C 180,E1 185.118,E2 185.118} C_VEL
LIN {X 0,Y 319.252,Z 1142.243,A -85,B 0,C 180,E1 183.771,E2 183.771} C_VEL
LIN {X 0,Y 338.107,Z 1121.054,A -85,B 0,C 180,E1 182.373,E2 182.373} C_VEL
LIN {X 0,Y 353.57,Z 1101.424,A -85,B 0,C 180,E1 181.345,E2 181.345} C_VEL
LIN {X 0,Y 366.424,Z 1083.396,A -85,B 0,C 180,E1 180.561,E2 180.561} C_VEL
LIN {X 0,Y 378.469,Z 1064.708,A -85,B 0,C 180,E1 179.888,E2 179.888} C_VEL
LIN {X 0,Y 379.146,Z 1063.608,A -85,B 0,C 180,E1 179.849,E2 179.849} C_VEL
LIN {X 0,Y 367.011,Z 1082.464,A -85,B 0,C 180,E1 179.146,E2 179.146} C_VEL
LIN {X 0,Y 354.12,Z 1100.544,A -85,B 0,C 180,E1 178.348,E2 178.348} C_VEL
LIN {X 0,Y 338.645,Z 1120.164,A -85,B 0,C 180,E1 177.292,E2 177.292} C_VEL
LIN {X 0,Y 319.809,Z 1141.321,A -85,B 0,C 180,E1 175.869,E2 175.869} C_VEL
LIN {X 0,Y 303.981,Z 1157.315,A -85,B 0,C 180,E1 174.526,E2 174.526} C_VEL
LIN {X 0,Y 288.123,Z 1171.975,A -85,B 0,C 180,E1 173.012,E2 173.012} C_VEL
LIN {X 0,Y 271.199,Z 1186.312,A -85,B 0,C 180,E1 171.172,E2 171.172} C_VEL
LIN {X 0,Y 249.984,Z 1202.643,A -85,B 0,C 180,E1 168.463,E2 168.463} C_VEL
LIN {X 0,Y 230.125,Z 1216.266,A -85,B 0,C 180,E1 165.403,E2 165.403} C_VEL
LIN {X 0,Y 213.158,Z 1226.96,A -85,B 0,C 180,E1 162.237,E2 162.237} C_VEL
LIN {X 0,Y 196.675,Z 1236.556,A -85,B 0,C 180,E1 158.508,E2 158.508} C_VEL
LIN {X 0,Y 176.835,Z 1247.287,A -85,B 0,C 180,E1 152.741,E2 152.741} C_VEL
LIN {X 0,Y 158.763,Z 1256.091,A -85,B 0,C 180,E1 145.606,E2 145.606} C_VEL
LIN {X 0,Y 145.71,Z 1262.196,A -85,B 0,C 180,E1 138.43,E2 138.43} C_VEL
LIN {X 0,Y 135.033,Z 1267.123,A -85,B 0,C 180,E1 130.12,E2 130.12} C_VEL
LIN {X 0,Y 126.022,Z 1271.536,A -85,B 0,C 180,E1 118.96,E2 118.96} C_VEL
LIN {X 0,Y 121.212,Z 1274.253,A -85,B 0,C 180,E1 106.795,E2 106.795} C_VEL
LIN {X 0,Y 120.032,Z 1275.36,A -85,B 0,C 180,E1 97.192,E2 97.192} C_VEL
LIN {X 0,Y 119.898,Z 1275.678,A -85,B 0,C 180,E1 89.536,E2 89.536} C_VEL
LIN {X 0,Y 120.074,Z 1275.327,A -85,B 0,C 180,E1 81.876,E2 81.876} C_VEL
LIN {X 0,Y 121.835,Z 1273.929,A -85,B 0,C 180,E1 70.7,E2 70.7} C_VEL
LIN {X 0,Y 127.37,Z 1270.822,A -85,B 0,C 180,E1 58.811,E2 58.811} C_VEL
LIN {X 0,Y 135.368,Z 1267.008,A -85,B 0,C 180,E1 49.476,E2 49.476} C_VEL
LIN {X 0,Y 146.143,Z 1262.053,A -85,B 0,C 180,E1 41.204,E2 41.204} C_VEL
LIN {X 0,Y 159.732,Z 1255.711,A -85,B 0,C 180,E1 33.857,E2 33.857} C_VEL
LIN {X 0,Y 178.766,Z 1246.335,A -85,B 0,C 180,E1 26.528,E2 26.528} C_VEL
LIN {X 0,Y 196.544,Z 1236.737,A -85,B 0,C 180,E1 21.441,E2 21.441} C_VEL
LIN {X 0,Y 213.03,Z 1227.158,A -85,B 0,C 180,E1 17.706,E2 17.706} C_VEL
LIN {X 0,Y 230.261,Z 1216.316,A -85,B 0,C 180,E1 14.491,E2 14.491} C_VEL
LIN {X 0,Y 250.828,Z 1202.219,A -85,B 0,C 180,E1 11.339,E2 11.339} C_VEL
LIN {X 0,Y 271.838,Z 1185.992,A -85,B 0,C 180,E1 8.674,E2 8.674} C_VEL
LIN {X 0,Y 288.023,Z 1172.292,A -85,B 0,C 180,E1 6.918,E2 6.918} C_VEL
LIN {X 0,Y 304.258,Z 1157.301,A -85,B 0,C 180,E1 5.369,E2 5.369} C_VEL
LIN {X 0,Y 321.412,Z 1139.935,A -85,B 0,C 180,E1 3.924,E2 3.924} C_VEL
LIN {X 0,Y 340.245,Z 1118.534,A -85,B 0,C 180,E1 2.515,E2 2.515} C_VEL
LIN {X 0,Y 354.452,Z 1100.484,A -85,B 0,C 180,E1 1.552,E2 1.552} C_VEL
LIN {X 0,Y 367.444,Z 1082.257,A -85,B 0,C 180,E1 0.75,E2 0.75} C_VEL
LIN {X 0,Y 378.557,Z 1065.037,A -85,B 0,C 180,E1 0.106,E2 0.106} C_VEL
LIN {X 0,Y 382.003,Z 1066.136,A -85,B 0,C 180,E1 -0.084,E2 -0.084} C_VEL
LIN {X 0,Y 382.003,Z 1110.356,A -85,B 0,C 180,E1 -0.084,E2 -0.084} C_VEL
LIN {X 0,Y 361.473,Z 1110.356,A -85,B 0,C 180,E1 0.279,E2 0.279} C_VEL
LIN {X 0,Y 359.487,Z 1108.356,A -85,B 0,C 180,E1 0.316,E2 0.316} C_VEL
LIN {X 0,Y 359.487,Z 1099.413,A -85,B 0,C 180,E1 0.316,E2 0.316} C_VEL
LIN {X 0,Y 356.124,Z 1098.17,A -85,B 0,C 180,E1 0.126,E2 0.126} C_VEL
LIN {X 0,Y 342.759,Z 1115.302,A -85,B 0,C 180,E1 -0.669,E2 -0.669} C_VEL
LIN {X 0,Y 327.671,Z 1132.882,A -85,B 0,C 180,E1 -1.665,E2 -1.665} C_VEL
LIN {X 0,Y 308.374,Z 1153.15,A -85,B 0,C 180,E1 -3.101,E2 -3.101} C_VEL
LIN {X 0,Y 289.888,Z 1170.375,A -85,B 0,C 180,E1 -4.671,E2 -4.671} C_VEL
LIN {X 0,Y 273.059,Z 1184.684,A -85,B 0,C 180,E1 -6.307,E2 -6.307} C_VEL
LIN {X 0,Y 256.522,Z 1197.577,A -85,B 0,C 180,E1 -8.151,E2 -8.151} C_VEL
LIN {X 0,Y 237.19,Z 1211.381,A -85,B 0,C 180,E1 -10.689,E2 -10.689} C_VEL
LIN {X 0,Y 213.743,Z 1226.37,A -85,B 0,C 180,E1 -14.496,E2 -14.496} C_VEL
LIN {X 0,Y 195.711,Z 1236.791,A -85,B 0,C 180,E1 -18.18,E2 -18.18} C_VEL
LIN {X 0,Y 179.389,Z 1245.5,A -85,B 0,C 180,E1 -22.323,E2 -22.323} C_VEL
LIN {X 0,Y 162.663,Z 1253.794,A -85,B 0,C 180,E1 -27.755,E2 -27.755} C_VEL
LIN {X 0,Y 143.843,Z 1262.494,A -85,B 0,C 180,E1 -36.283,E2 -36.283} C_VEL
LIN {X 0,Y 130.567,Z 1268.306,A -85,B 0,C 180,E1 -45.228,E2 -45.228} C_VEL
LIN {X 0,Y 121.658,Z 1272.284,A -85,B 0,C 180,E1 -54.319,E2 -54.319} C_VEL
LIN {X 0,Y 115.673,Z 1275.225,A -85,B 0,C 180,E1 -64.41,E2 -64.41} C_VEL
LIN {X 0,Y 112.697,Z 1277.076,A -85,B 0,C 180,E1 -74.579,E2 -74.579} C_VEL
LIN {X 0,Y 111.955,Z 1277.933,A -85,B 0,C 180,E1 -83.348,E2 -83.348} C_VEL
LIN {X 0,Y 111.896,Z 1278.184,A -85,B 0,C 180,E1 -91.039,E2 -91.039} C_VEL
LIN {X 0,Y 112.032,Z 1277.806,A -85,B 0,C 180,E1 -99.259,E2 -99.259} C_VEL
LIN {X 0,Y 113.854,Z 1276.349,A -85,B 0,C 180,E1 -110.581,E2 -110.581} C_VEL
LIN {X 0,Y 119.977,Z 1273.054,A -85,B 0,C 180,E1 -123.385,E2 -123.385} C_VEL
LIN {X 0,Y 128.685,Z 1269.089,A -85,B 0,C 180,E1 -133.154,E2 -133.154} C_VEL
LIN {X 0,Y 139.691,Z 1264.228,A -85,B 0,C 180,E1 -141.295,E2 -141.295} C_VEL
LIN {X 0,Y 152.9,Z 1258.276,A -85,B 0,C 180,E1 -148.242,E2 -148.242} C_VEL
LIN {X 0,Y 170.128,Z 1250.122,A -85,B 0,C 180,E1 -154.854,E2 -154.854} C_VEL
LIN {X 0,Y 191.586,Z 1238.973,A -85,B 0,C 180,E1 -160.864,E2 -160.864} C_VEL
LIN {X 0,Y 209.421,Z 1228.815,A -85,B 0,C 180,E1 -164.698,E2 -164.698} C_VEL
LIN {X 0,Y 226.228,Z 1218.43,A -85,B 0,C 180,E1 -167.65,E2 -167.65} C_VEL
LIN {X 0,Y 244.711,Z 1205.999,A -85,B 0,C 180,E1 -170.356,E2 -170.356} C_VEL
LIN {X 0,Y 266.952,Z 1189.454,A -85,B 0,C 180,E1 -173.044,E2 -173.044} C_VEL
LIN {X 0,Y 286.077,Z 1173.497,A -85,B 0,C 180,E1 -174.989,E2 -174.989} C_VEL
LIN {X 0,Y 301.901,Z 1159.053,A -85,B 0,C 180,E1 -176.392,E2 -176.392} C_VEL
LIN {X 0,Y 317.257,Z 1143.76,A -85,B 0,C 180,E1 -177.597,E2 -177.597} C_VEL
LIN {X 0,Y 333.061,Z 1126.508,A -85,B 0,C 180,E1 -178.706,E2 -178.706} C_VEL
LIN {X 0,Y 351.973,Z 1103.339,A -85,B 0,C 180,E1 -179.896,E2 -179.896} C_VEL
LIN {X 0,Y 356.706,Z 1097,A -85,B 0,C 180,E1 -180.171,E2 -180.171} C_VEL
LIN {X 0,Y 343.028,Z 1114.55,A -85,B 0,C 180,E1 -181.011,E2 -181.011} C_VEL
LIN {X 0,Y 328.671,Z 1131.289,A -85,B 0,C 180,E1 -181.971,E2 -181.971} C_VEL
LIN {X 0,Y 311.482,Z 1149.489,A -85,B 0,C 180,E1 -183.257,E2 -183.257} C_VEL
LIN {X 0,Y 291.087,Z 1168.705,A -85,B 0,C 180,E1 -184.993,E2 -184.993} C_VEL
LIN {X 0,Y 273.542,Z 1183.586,A -85,B 0,C 180,E1 -186.717,E2 -186.717} C_VEL
LIN {X 0,Y 256.873,Z 1196.519,A -85,B 0,C 180,E1 -188.595,E2 -188.595} C_VEL
LIN {X 0,Y 239.305,Z 1209.011,A -85,B 0,C 180,E1 -190.895,E2 -190.895} C_VEL
LIN {X 0,Y 217.364,Z 1223.195,A -85,B 0,C 180,E1 -194.383,E2 -194.383} C_VEL
LIN {X 0,Y 197.106,Z 1234.83,A -85,B 0,C 180,E1 -198.427,E2 -198.427} C_VEL
LIN {X 0,Y 180.785,Z 1243.453,A -85,B 0,C 180,E1 -202.518,E2 -202.518} C_VEL
LIN {X 0,Y 164.755,Z 1251.3,A -85,B 0,C 180,E1 -207.601,E2 -207.601} C_VEL
LIN {X 0,Y 148.258,Z 1258.879,A -85,B 0,C 180,E1 -214.618,E2 -214.618} C_VEL
LIN {X 0,Y 131.968,Z 1265.868,A -85,B 0,C 180,E1 -224.801,E2 -224.801} C_VEL
LIN {X 0,Y 122.529,Z 1269.903,A -85,B 0,C 180,E1 -234.002,E2 -234.002} C_VEL
LIN {X 0,Y 116.263,Z 1272.787,A -85,B 0,C 180,E1 -243.97,E2 -243.97} C_VEL
LIN {X 0,Y 112.994,Z 1274.606,A -85,B 0,C 180,E1 -254.064,E2 -254.064} C_VEL
LIN {X 0,Y 112.007,Z 1275.491,A -85,B 0,C 180,E1 -263.321,E2 -263.321} C_VEL
LIN {X 0,Y 111.896,Z 1275.743,A -85,B 0,C 180,E1 -271.009,E2 -271.009} C_VEL
LIN {X 0,Y 112.122,Z 1275.394,A -85,B 0,C 180,E1 -279.222,E2 -279.222} C_VEL
LIN {X 0,Y 114.26,Z 1273.949,A -85,B 0,C 180,E1 -291.009,E2 -291.009} C_VEL
LIN {X 0,Y 120.382,Z 1270.912,A -85,B 0,C 180,E1 -303.225,E2 -303.225} C_VEL
LIN {X 0,Y 129.156,Z 1267.099,A -85,B 0,C 180,E1 -312.923,E2 -312.923} C_VEL
LIN {X 0,Y 140.636,Z 1262.205,A -85,B 0,C 180,E1 -321.269,E2 -321.269} C_VEL
LIN {X 0,Y 154.747,Z 1256.01,A -85,B 0,C 180,E1 -328.504,E2 -328.504} C_VEL
LIN {X 0,Y 173.973,Z 1247.055,A -85,B 0,C 180,E1 -335.555,E2 -335.555} C_VEL
LIN {X 0,Y 193.638,Z 1236.828,A -85,B 0,C 180,E1 -340.868,E2 -340.868} C_VEL
LIN {X 0,Y 210.634,Z 1227.248,A -85,B 0,C 180,E1 -344.465,E2 -344.465} C_VEL
LIN {X 0,Y 228.313,Z 1216.406,A -85,B 0,C 180,E1 -347.54,E2 -347.54} C_VEL
LIN {X 0,Y 249.323,Z 1202.309,A -85,B 0,C 180,E1 -350.54,E2 -350.54} C_VEL
LIN {X 0,Y 269.95,Z 1186.693,A -85,B 0,C 180,E1 -352.983,E2 -352.983} C_VEL
LIN {X 0,Y 287.142,Z 1172.38,A -85,B 0,C 180,E1 -354.724,E2 -354.724} C_VEL
LIN {X 0,Y 303.596,Z 1157.388,A -85,B 0,C 180,E1 -356.185,E2 -356.185} C_VEL
LIN {X 0,Y 320.297,Z 1140.696,A -85,B 0,C 180,E1 -357.495,E2 -357.495} C_VEL
LIN {X 0,Y 339.984,Z 1118.62,A -85,B 0,C 180,E1 -358.866,E2 -358.866} C_VEL
LIN {X 0,Y 354.368,Z 1100.512,A -85,B 0,C 180,E1 -359.771,E2 -359.771} C_VEL
LIN {X 0,Y 356.124,Z 1098.17,A -85,B 0,C 180,E1 -359.874,E2 -359.874} C_VEL
LIN {X 0,Y 349.335,Z 1107.235,A -85,B 0,C 180,E1 -360.111,E2 -360.111} C_VEL
LIN {X 0,Y 340.787,Z 1117.635,A -85,B 0,C 180,E1 -360.066,E2 -360.066} C_VEL
LIN {X 0,Y 331.515,Z 1128.377,A -85,B 0,C 180,E1 -359.705,E2 -359.705} C_VEL
LIN {X 0,Y 325.632,Z 1134.876,A -85,B 0,C 180,E1 -359.35,E2 -359.35} C_VEL
LIN {X 0,Y 305.128,Z 1155.632,A -85,B 0,C 180,E1 -357.895,E2 -357.895} C_VEL
LIN {X 0,Y 288.45,Z 1170.785,A -85,B 0,C 180,E1 -356.542,E2 -356.542} C_VEL
LIN {X 0,Y 271.953,Z 1184.482,A -85,B 0,C 180,E1 -355.024,E2 -355.024} C_VEL
LIN {X 0,Y 254.715,Z 1197.568,A -85,B 0,C 180,E1 -353.214,E2 -353.214} C_VEL
LIN {X 0,Y 233.123,Z 1212.492,A -85,B 0,C 180,E1 -350.513,E2 -350.513} C_VEL
LIN {X 0,Y 211.186,Z 1225.83,A -85,B 0,C 180,E1 -347.142,E2 -347.142} C_VEL
LIN {X 0,Y 193.639,Z 1235.552,A -85,B 0,C 180,E1 -343.79,E2 -343.79} C_VEL
LIN {X 0,Y 176.802,Z 1244.108,A -85,B 0,C 180,E1 -339.816,E2 -339.816} C_VEL
LIN {X 0,Y 159.4,Z 1252.236,A -85,B 0,C 180,E1 -334.564,E2 -334.564} C_VEL
LIN {X 0,Y 139.551,Z 1260.729,A -85,B 0,C 180,E1 -326.191,E2 -326.191} C_VEL
LIN {X 0,Y 125.267,Z 1266.376,A -85,B 0,C 180,E1 -317.23,E2 -317.23} C_VEL
LIN {X 0,Y 115.452,Z 1270.218,A -85,B 0,C 180,E1 -307.925,E2 -307.925} C_VEL
LIN {X 0,Y 108.633,Z 1273.037,A -85,B 0,C 180,E1 -297.382,E2 -297.382} C_VEL
LIN {X 0,Y 105.058,Z 1274.791,A -85,B 0,C 180,E1 -286.573,E2 -286.573} C_VEL
LIN {X 0,Y 104.024,Z 1275.589,A -85,B 0,C 180,E1 -277.162,E2 -277.162} C_VEL
LIN {X 0,Y 103.903,Z 1275.821,A -85,B 0,C 180,E1 -268.881,E2 -268.881} C_VEL
LIN {X 0,Y 104.171,Z 1275.472,A -85,B 0,C 180,E1 -260.035,E2 -260.035} C_VEL
LIN {X 0,Y 106.519,Z 1274.095,A -85,B 0,C 180,E1 -247.931,E2 -247.931} C_VEL
LIN {X 0,Y 113.619,Z 1270.934,A -85,B 0,C 180,E1 -234.476,E2 -234.476} C_VEL
LIN {X 0,Y 123.286,Z 1267.103,A -85,B 0,C 180,E1 -224.446,E2 -224.446} C_VEL
LIN {X 0,Y 135.201,Z 1262.381,A -85,B 0,C 180,E1 -216.265,E2 -216.265} C_VEL
LIN {X 0,Y 149.837,Z 1256.321,A -85,B 0,C 180,E1 -209.153,E2 -209.153} C_VEL
LIN {X 0,Y 169.65,Z 1247.546,A -85,B 0,C 180,E1 -202.263,E2 -202.263} C_VEL
LIN {X 0,Y 190.32,Z 1237.197,A -85,B 0,C 180,E1 -197.004,E2 -197.004} C_VEL
LIN {X 0,Y 207.77,Z 1227.658,A -85,B 0,C 180,E1 -193.539,E2 -193.539} C_VEL
LIN {X 0,Y 224.928,Z 1217.422,A -85,B 0,C 180,E1 -190.732,E2 -190.732} C_VEL
LIN {X 0,Y 243.479,Z 1205.318,A -85,B 0,C 180,E1 -188.198,E2 -188.198} C_VEL
LIN {X 0,Y 266.268,Z 1188.797,A -85,B 0,C 180,E1 -185.624,E2 -185.624} C_VEL
LIN {X 0,Y 285.606,Z 1173.003,A -85,B 0,C 180,E1 -183.783,E2 -183.783} C_VEL
LIN {X 0,Y 302.247,Z 1158.068,A -85,B 0,C 180,E1 -182.405,E2 -182.405} C_VEL
LIN {X 0,Y 318.549,Z 1142.012,A -85,B 0,C 180,E1 -181.213,E2 -181.213} C_VEL
LIN {X 0,Y 333.977,Z 1125.3,A -85,B 0,C 180,E1 -180.185,E2 -180.185} C_VEL
LIN {X 0,Y 318.012,Z 1142.648,A -85,B 0,C 180,E1 -179.161,E2 -179.161} C_VEL
LIN {X 0,Y 302.162,Z 1158.329,A -85,B 0,C 180,E1 -178.016,E2 -178.016} C_VEL
LIN {X 0,Y 286.448,Z 1172.554,A -85,B 0,C 180,E1 -176.736,E2 -176.736} C_VEL
LIN {X 0,Y 269.925,Z 1186.262,A -85,B 0,C 180,E1 -175.218,E2 -175.218} C_VEL
LIN {X 0,Y 248.87,Z 1202.196,A -85,B 0,C 180,E1 -172.951,E2 -172.951} C_VEL
LIN {X 0,Y 227.113,Z 1216.751,A -85,B 0,C 180,E1 -170.113,E2 -170.113} C_VEL
LIN {X 0,Y 209.147,Z 1227.684,A -85,B 0,C 180,E1 -167.258,E2 -167.258} C_VEL
LIN {X 0,Y 191.568,Z 1237.491,A -85,B 0,C 180,E1 -163.841,E2 -163.841} C_VEL
LIN {X 0,Y 173.137,Z 1246.924,A -85,B 0,C 180,E1 -159.34,E2 -159.34} C_VEL
LIN {X 0,Y 150.797,Z 1257.262,A -85,B 0,C 180,E1 -151.888,E2 -151.888} C_VEL
LIN {X 0,Y 135.857,Z 1263.62,A -85,B 0,C 180,E1 -144.797,E2 -144.797} C_VEL
LIN {X 0,Y 123.643,Z 1268.622,A -85,B 0,C 180,E1 -136.576,E2 -136.576} C_VEL
LIN {X 0,Y 114.26,Z 1272.474,A -85,B 0,C 180,E1 -127.16,E2 -127.16} C_VEL
LIN {X 0,Y 107.845,Z 1275.336,A -85,B 0,C 180,E1 -116.441,E2 -116.441} C_VEL
LIN {X 0,Y 104.596,Z 1277.178,A -85,B 0,C 180,E1 -104.973,E2 -104.973} C_VEL
LIN {X 0,Y 103.929,Z 1277.91,A -85,B 0,C 180,E1 -95.537,E2 -95.537} C_VEL
LIN {X 0,Y 103.907,Z 1278.056,A -85,B 0,C 180,E1 -87.81,E2 -87.81} C_VEL
LIN {X 0,Y 104.136,Z 1277.673,A -85,B 0,C 180,E1 -78.945,E2 -78.945} C_VEL
LIN {X 0,Y 106.766,Z 1275.949,A -85,B 0,C 180,E1 -66.271,E2 -66.271} C_VEL
LIN {X 0,Y 113.488,Z 1272.845,A -85,B 0,C 180,E1 -53.841,E2 -53.841} C_VEL
LIN {X 0,Y 122.702,Z 1269.055,A -85,B 0,C 180,E1 -44.206,E2 -44.206} C_VEL
LIN {X 0,Y 134.572,Z 1264.207,A -85,B 0,C 180,E1 -35.94,E2 -35.94} C_VEL
LIN {X 0,Y 148.842,Z 1258.172,A -85,B 0,C 180,E1 -28.926,E2 -28.926} C_VEL
LIN {X 0,Y 166.68,Z 1250.135,A -85,B 0,C 180,E1 -22.541,E2 -22.541} C_VEL
LIN {X 0,Y 188.951,Z 1239.014,A -85,B 0,C 180,E1 -16.741,E2 -16.741} C_VEL
LIN {X 0,Y 207.313,Z 1228.873,A -85,B 0,C 180,E1 -13.074,E2 -13.074} C_VEL
LIN {X 0,Y 224.641,Z 1218.442,A -85,B 0,C 180,E1 -10.256,E2 -10.256} C_VEL
LIN {X 0,Y 242.557,Z 1206.674,A -85,B 0,C 180,E1 -7.819,E2 -7.819} C_VEL
LIN {X 0,Y 264.094,Z 1191.146,A -85,B 0,C 180,E1 -5.384,E2 -5.384} C_VEL
LIN {X 0,Y 284.718,Z 1174.29,A -85,B 0,C 180,E1 -3.423,E2 -3.423} C_VEL
LIN {X 0,Y 301.12,Z 1159.569,A -85,B 0,C 180,E1 -2.073,E2 -2.073} C_VEL
LIN {X 0,Y 317.237,Z 1143.727,A -85,B 0,C 180,E1 -0.903,E2 -0.903} C_VEL
LIN {X 0,Y 333.369,Z 1126.296,A -85,B 0,C 180,E1 0.153,E2 0.153} C_VEL
LIN {X 0,Y 325.632,Z 1134.876,A -85,B 0,C 180,E1 0.65,E2 0.65} C_VEL
LIN {X 0,Y 321.129,Z 1139.739,A -85,B 0,C 180,E1 0.786,E2 0.786} C_VEL
LIN {X 0,Y 314.906,Z 1146.09,A -85,B 0,C 180,E1 0.591,E2 0.591} C_VEL
LIN {X 0,Y 300.565,Z 1159.826,A -85,B 0,C 180,E1 -0.522,E2 -0.522} C_VEL
LIN {X 0,Y 282.087,Z 1176.142,A -85,B 0,C 180,E1 -1.932,E2 -1.932} C_VEL
